DATA_BLOCK "DB23_AlarmProgram"   // DB23
{ S7_Optimized_Access := 'FALSE' }
AUTHOR : Robopac
VERSION : 0.0
// stored: AutoNumber false, IsOnlyStoredInLoadMemory false, IsWriteProtectedInAS false
   VAR RETAIN
      dbx0_0 : Bool := FALSE;   // Alarm 1: Pressure switch (Technoplat)
      dbx0_1 : Bool := FALSE;   // Alarm 2: Door open request (Technoplat)
      dbx0_2 : Bool := FALSE;   // Alarm 3: Emergency push button (Technoplat)
      dbx0_3 : Bool := FALSE;   // Alarm 4: Thermic alarm (Technoplat)
      dbx0_4 : Bool := FALSE;   // Alarm 5: Fault inverters (Technoplat)
      dbx0_5 : Bool := FALSE;   // Alarm 6: Motor start missing (Technoplat)
      dbx0_6 : Bool := FALSE;   // Alarm 7: Stop cycle by operator (Technoplat)
      dbx0_7 : Bool := FALSE;   // Alarm 8: Film ended or broken (Technoplat)
      dbx1_0 : Bool := FALSE;   // Alarm 9: Machine table not in phase (Technoplat)
      dbx1_1 : Bool := FALSE;   // Alarm 10: The spool carriage encoder is not running (Technoplat)
      dbx1_2 : Bool := FALSE;   // Alarm 11: Table encoder not working well
      dbx1_3 : Bool := FALSE;   // Alarm 12: Overspeed for table rotation (Technoplat)
      dbx1_4 : Bool := FALSE;   // Alarm 13: Phase table sensor lost (Technoplat)
      dbx1_5 : Bool := FALSE;   // Alarm 14: table deceleration not correct (Technoplat)
      dbx1_6 : Bool := FALSE;   // Alarm 15: Pressure plate not up (Pressure plate)
      dbx1_7 : Bool := FALSE;   // Alarm 16: Timeout for pressure plate upward/downward (Pressure plate)
      dbx2_0 : Bool := FALSE;   // Alarm 17: Pallet lifter not down (Lifter)
      dbx2_1 : Bool := FALSE;   // Alarm 18: Timeout for pallet lifter upward/downward (Lifter)
      dbx2_2 : Bool := FALSE;   // Alarm 19: Wrong data program for the pallet on the machine (Technoplat)
      dbx2_3 : Bool := FALSE;   // Alarm 20: Sysdata error (Technoplat)
      dbx2_4 : Bool := FALSE;   // Alarm 21: Spool carriage not down (Technoplat)
      dbx2_5 : Bool := FALSE;   // Alarm 22: Pressure plate positioning lost during rotation
      dbx2_6 : Bool := FALSE;   // Alarm 23:
      dbx2_7 : Bool := FALSE;   // Alarm 24: Emergency on infeed safety barrier (Barrier)
      dbx3_0 : Bool := FALSE;   // Alarm 25: Emergency on outfeed safety barrier (Barrier)
      dbx3_1 : Bool := FALSE;   // Alarm 26: Safety barrier excluded in automatic mode (Barrier)
      dbx3_2 : Bool := FALSE;   // Alarm 27: Timeout for rope unit open/close (Rope unit)
      dbx3_3 : Bool := FALSE;   // Alarm 28: Timeout for full rope unit open/close (Rope unit)
      dbx3_4 : Bool := FALSE;   // Alarm 29:
      dbx3_5 : Bool := FALSE;   // Alarm 30: Profinet communication error
      dbx3_6 : Bool := FALSE;   // Alarm 31: Modbus communication error
      dbx3_7 : Bool := FALSE;   // Alarm 32:
      dbx4_0 : Bool := FALSE;   // Alarm 33: Pallet positioning released during table rotation (Conveyor
      dbx4_1 : Bool := FALSE;   // Alarm 34: Pallet in transit in infeed (Conveyor)
      dbx4_2 : Bool := FALSE;   // Alarm 35: Pallet in transit in outfeed (Conveyor)
      dbx4_3 : Bool := FALSE;   // Alarm 36: Wrong pallet positioning (Conveyor)
      dbx4_4 : Bool := FALSE;   // Alarm 37: Infeed ring rotation control engaged (Conveyor)
      dbx4_5 : Bool := FALSE;   // Alarm 38: Outfeed ring rotation control engaged (Conveyor)
      dbx4_6 : Bool := FALSE;   // Alarm 39: Technoplat table not in load phase
      dbx4_7 : Bool := FALSE;   // Alarm 40: Technoplat table not in unload phase
      dbx5_0 : Bool := FALSE;   // Alarm 41: Contrast carriage not back
      dbx5_1 : Bool := FALSE;   // Alarm 42: Timeout contrast carriage forward/backward
      dbx5_2 : Bool := FALSE;   // Alarm 43: Clamp not closed (Clamp)
      dbx5_3 : Bool := FALSE;   // Alarm 44: Welder contrast not down (Clamp)
      dbx5_4 : Bool := FALSE;   // Alarm 45: Welder unit not down (Clamp)
      dbx5_5 : Bool := FALSE;   // Alarm 46: Clamp not down (Clamp)
      dbx5_6 : Bool := FALSE;   // Alarm 47: Welder contrast not up (Clamp)
      dbx5_7 : Bool := FALSE;   // Alarm 48: Timeout for clamp open/close (Clamp)
      dbx6_0 : Bool := FALSE;   // Alarm 49: Timeout for clamp upward/downward (Clamp)
      dbx6_1 : Bool := FALSE;   // Alarm 50: Timeout for welder contrast upward/downward (Clamp)
      dbx6_2 : Bool := FALSE;   // Alarm 51: Timeout for welder unit upward/downward (Clamp)
      dbx6_3 : Bool := FALSE;   // Alarm 52: Check the welder circuit (Clamp)
      dbx6_4 : Bool := FALSE;   // Alarm 53: Welder and cut unit not backward (Clamp)
      dbx6_5 : Bool := FALSE;   // Alarm 54: Timeout for welder and cut unit forward/backward (Clamp)
      dbx6_6 : Bool := FALSE;   // Alarm 55: Timeout for clamp carriage forward/backward (Clamp)
      dbx6_7 : Bool := FALSE;   // Alarm 56: Clamp carriage not backward (Clamp)
      dbx7_0 : Bool := FALSE;   // Alarm 57: Top carriage not up (Top)
      dbx7_1 : Bool := FALSE;   // Alarm 58: Top carriage not backward (Top)
      dbx7_2 : Bool := FALSE;   // Alarm 59: Top cutter not backward (Top)
      dbx7_3 : Bool := FALSE;   // Alarm 60: Clamp to pull top film not open (Top)
      dbx7_4 : Bool := FALSE;   // Alarm 61: Clamp to block top film not closed (Top)
      dbx7_5 : Bool := FALSE;   // Alarm 62: Top carriage not in position (Top)
      dbx7_6 : Bool := FALSE;   // Alarm 63: Top carriage not inside top film cut area (Top)
      dbx7_7 : Bool := FALSE;   // Alarm 64: Safety for top carriage position (Top)
      dbx8_0 : Bool := FALSE;   // Alarm 65: Timeout for top cutter (Top)
      dbx8_1 : Bool := FALSE;   // Alarm 66: Timeout for clamp to pull top film (Top)
      dbx8_2 : Bool := FALSE;   // Alarm 67: Timeout for clamp to block top film (Top)
      dbx8_3 : Bool := FALSE;   // Alarm 68: Top film ended or broken (Top)
      dbx8_4 : Bool := FALSE;   // Alarm 69: Infeed safety for top carriage up/down (Top)
      dbx8_5 : Bool := FALSE;   // Alarm 70: Outfeed safety for top carriage up/down (Top)
      dbx8_6 : Bool := FALSE;   // Alarm 71: Clamp to blok top film not open (Top)
      dbx8_7 : Bool := FALSE;   // Alarm 72: Top rele' brake broken (Top)
      dbx9_0 : Bool := FALSE;   // Alarm 73: Top not in position (Top inside signal)
      dbx9_1 : Bool := FALSE;   // Alarm 74: LIFTER POS.2 EXTRASTROKE UP
      dbx9_2 : Bool := FALSE;   // Alarm 75: LIFTER POS.2 FOOT SAFETY
      dbx9_3 : Bool := FALSE;   // Alarm 76: LIFTER POS.2 TIMEOUT CONVEYOR
      dbx9_4 : Bool := FALSE;   // Alarm 77: LIFTER POS.2 TIMEOUT UPSTROKE
      dbx9_5 : Bool := FALSE;   // Alarm 78: LIFTER POS.2 TIMEOUT DOWNSTROKE
      dbx9_6 : Bool := FALSE;   // Alarm 79: LABEL FAULT
      dbx9_7 : Bool := FALSE;   // Alarm 80: Label not in home position with table rotation
      dbx10_0 : Bool := FALSE;   // Alarm 81: Fire door not open during pallet transit
      dbx10_1 : Bool := FALSE;   // Alarm 82:
      dbx10_2 : Bool := FALSE;   // Alarm 83:
      dbx10_3 : Bool := FALSE;   // Alarm 84:
      dbx10_4 : Bool := FALSE;   // Alarm 85:
      dbx10_5 : Bool := FALSE;   // Alarm 86:
      dbx10_6 : Bool := FALSE;   // Alarm 87:
      dbx10_7 : Bool := FALSE;   // Alarm 88:
      dbx11_0 : Bool := FALSE;   // Alarm 89:
      dbx11_1 : Bool := FALSE;   // Alarm 90:
      dbx11_2 : Bool := FALSE;   // Alarm 91:
      dbx11_3 : Bool := FALSE;   // Alarm 92:
      dbx11_4 : Bool := FALSE;   // Alarm 93:
      dbx11_5 : Bool := FALSE;   // Alarm 94:
      dbx11_6 : Bool := FALSE;   // Alarm 95:
      dbx11_7 : Bool := FALSE;   // Alarm 96:
      dbx12_0 : Bool := FALSE;   // Alarm 97:
      dbx12_1 : Bool := FALSE;   // Alarm 98:
      dbx12_2 : Bool := FALSE;   // Alarm 99:
      dbx12_3 : Bool := FALSE;   // Alarm 100:
      dbx12_4 : Bool := FALSE;   // Alarm 101:
      dbx12_5 : Bool := FALSE;   // Alarm 102:
      dbx12_6 : Bool := FALSE;   // Alarm 103:
      dbx12_7 : Bool := FALSE;   // Alarm 104:
      dbx13_0 : Bool := FALSE;   // Alarm 105:
      dbx13_1 : Bool := FALSE;   // Alarm 106:
      dbx13_2 : Bool := FALSE;   // Alarm 107:
      dbx13_3 : Bool := FALSE;   // Alarm 108:
      dbx13_4 : Bool := FALSE;   // Alarm 109:
      dbx13_5 : Bool := FALSE;   // Alarm 110:
      dbx13_6 : Bool := FALSE;   // Alarm 111:
      dbx13_7 : Bool := FALSE;   // Alarm 112:
      dbx14_0 : Bool := FALSE;   // Alarm 113:
      dbx14_1 : Bool := FALSE;   // Alarm 114:
      dbx14_2 : Bool := FALSE;   // Alarm 115:
      dbx14_3 : Bool := FALSE;   // Alarm 116:
      dbx14_4 : Bool := FALSE;   // Alarm 117:
      dbx14_5 : Bool := FALSE;   // Alarm 118:
      dbx14_6 : Bool := FALSE;   // Alarm 119:
      dbx14_7 : Bool := FALSE;   // Alarm 120:
      dbx15_0 : Bool := FALSE;   // Alarm 121:
      dbx15_1 : Bool := FALSE;   // Alarm 122:
      dbx15_2 : Bool := FALSE;   // Alarm 123:
      dbx15_3 : Bool := FALSE;   // Alarm 124:
      dbx15_4 : Bool := FALSE;   // Alarm 125:
      dbx15_5 : Bool := FALSE;   // Alarm 126:
      dbx15_6 : Bool := FALSE;   // Alarm 127:
      dbx15_7 : Bool := FALSE;   // Alarm 128:
      dbx16_0 : Bool := FALSE;   // Alarm 129:
      dbx16_1 : Bool := FALSE;   // Alarm 130:
      dbx16_2 : Bool := FALSE;   // Alarm 131:
      dbx16_3 : Bool := FALSE;   // Alarm 132:
      dbx16_4 : Bool := FALSE;   // Alarm 133:
      dbx16_5 : Bool := FALSE;   // Alarm 134:
      dbx16_6 : Bool := FALSE;   // Alarm 135:
      dbx16_7 : Bool := FALSE;   // Alarm 136:
      dbx17_0 : Bool := FALSE;   // Alarm 137:
      dbx17_1 : Bool := FALSE;   // Alarm 138:
      dbx17_2 : Bool := FALSE;   // Alarm 139:
      dbx17_3 : Bool := FALSE;   // Alarm 140:
      dbx17_4 : Bool := FALSE;   // Alarm 141:
      dbx17_5 : Bool := FALSE;   // Alarm 142:
      dbx17_6 : Bool := FALSE;   // Alarm 143:
      dbx17_7 : Bool := FALSE;   // Alarm 144:
      dbx18_0 : Bool := FALSE;   // Alarm 145:
      dbx18_1 : Bool := FALSE;   // Alarm 146:
      dbx18_2 : Bool := FALSE;   // Alarm 147:
      dbx18_3 : Bool := FALSE;   // Alarm 148:
      dbx18_4 : Bool := FALSE;   // Alarm 149:
      dbx18_5 : Bool := FALSE;   // Alarm 150:
      dbx18_6 : Bool := FALSE;   // Alarm 151:
      dbx18_7 : Bool := FALSE;   // Alarm 152:
      dbx19_0 : Bool := FALSE;   // Alarm 153:
      dbx19_1 : Bool := FALSE;   // Alarm 154:
      dbx19_2 : Bool := FALSE;   // Alarm 155:
      dbx19_3 : Bool := FALSE;   // Alarm 156:
      dbx19_4 : Bool := FALSE;   // Alarm 157:
      dbx19_5 : Bool := FALSE;   // Alarm 158:
      dbx19_6 : Bool := FALSE;   // Alarm 159:
      dbx19_7 : Bool := FALSE;   // Alarm 160:
      dbx20_0 : Bool := FALSE;   // Alarm 161:
      dbx20_1 : Bool := FALSE;   // Alarm 162:
      dbx20_2 : Bool := FALSE;   // Alarm 163:
      dbx20_3 : Bool := FALSE;   // Alarm 164:
      dbx20_4 : Bool := FALSE;   // Alarm 165:
      dbx20_5 : Bool := FALSE;   // Alarm 166:
      dbx20_6 : Bool := FALSE;   // Alarm 167:
      dbx20_7 : Bool := FALSE;   // Alarm 168:
      dbx21_0 : Bool := FALSE;   // Alarm 169:
      dbx21_1 : Bool := FALSE;   // Alarm 170:
      dbx21_2 : Bool := FALSE;   // Alarm 171:
      dbx21_3 : Bool := FALSE;   // Alarm 172:
      dbx21_4 : Bool := FALSE;   // Alarm 173:
      dbx21_5 : Bool := FALSE;   // Alarm 174:
      dbx21_6 : Bool := FALSE;   // Alarm 175:
      dbx21_7 : Bool := FALSE;   // Alarm 176:
      dbx22_0 : Bool := FALSE;   // Alarm 177:
      dbx22_1 : Bool := FALSE;   // Alarm 178:
      dbx22_2 : Bool := FALSE;   // Alarm 179:
      dbx22_3 : Bool := FALSE;   // Alarm 180:
      dbx22_4 : Bool := FALSE;   // Alarm 181:
      dbx22_5 : Bool := FALSE;   // Alarm 182:
      dbx22_6 : Bool := FALSE;   // Alarm 183:
      dbx22_7 : Bool := FALSE;   // Alarm 184:
      dbx23_0 : Bool := FALSE;   // Alarm 185:
      dbx23_1 : Bool := FALSE;   // Alarm 186:
      dbx23_2 : Bool := FALSE;   // Alarm 187:
      dbx23_3 : Bool := FALSE;   // Alarm 188:
      dbx23_4 : Bool := FALSE;   // Alarm 189:
      dbx23_5 : Bool := FALSE;   // Alarm 190:
      dbx23_6 : Bool := FALSE;   // Alarm 191:
      dbx23_7 : Bool := FALSE;   // Alarm 192:
      dbx24_0 : Bool := FALSE;   // Alarm 193:
      dbx24_1 : Bool := FALSE;   // Alarm 194:
      dbx24_2 : Bool := FALSE;   // Alarm 195:
      dbx24_3 : Bool := FALSE;   // Alarm 196:
      dbx24_4 : Bool := FALSE;   // Alarm 197:
      dbx24_5 : Bool := FALSE;   // Alarm 198:
      dbx24_6 : Bool := FALSE;   // Alarm 199:
      dbx24_7 : Bool := FALSE;   // Alarm 200:
      dbx25_0 : Bool := FALSE;   // Alarm 201:
      dbx25_1 : Bool := FALSE;   // Alarm 202:
      dbx25_2 : Bool := FALSE;   // Alarm 203:
      dbx25_3 : Bool := FALSE;   // Alarm 204:
      dbx25_4 : Bool := FALSE;   // Alarm 205:
      dbx25_5 : Bool := FALSE;   // Alarm 206:
      dbx25_6 : Bool := FALSE;   // Alarm 207:
      dbx25_7 : Bool := FALSE;   // Alarm 208:
      dbx26_0 : Bool := FALSE;   // Warning 1: %10 Prestretch film on spool carriage (Technoplat)
      dbx26_1 : Bool := FALSE;   // Warning 2:
      dbx26_2 : Bool := FALSE;   // Warning 3: Request to reset encoder on spool carriage (Technoplat)
      dbx26_3 : Bool := FALSE;   // Warning 4:
      dbx26_4 : Bool := FALSE;   // Warning 5: Request to reset encoder on table rotation (Technoplat)
      dbx26_5 : Bool := FALSE;   // Warning 6:
      dbx26_6 : Bool := FALSE;   // Warning 7:
      dbx26_7 : Bool := FALSE;   // Warning 8: Fire door closing request
      dbx27_0 : Bool := FALSE;   // Warning 9: Timeout for door opening
      dbx27_1 : Bool := FALSE;   // Warning 10:
      dbx27_2 : Bool := FALSE;   // Warning 11:
      dbx27_3 : Bool := FALSE;   // Warning 12:
      dbx27_4 : Bool := FALSE;   // Warning 13:
      dbx27_5 : Bool := FALSE;   // Warning 14:
      dbx27_6 : Bool := FALSE;   // Warning 15:
      dbx27_7 : Bool := FALSE;   // Warning 16:
      dbx28_0 : Bool := FALSE;   // Warning 17:
      dbx28_1 : Bool := FALSE;   // Warning 18:
      dbx28_2 : Bool := FALSE;   // Warning 19:
      dbx28_3 : Bool := FALSE;   // Warning 20:
      dbx28_4 : Bool := FALSE;   // Warning 21:
      dbx28_5 : Bool := FALSE;   // Warning 22:
      dbx28_6 : Bool := FALSE;   // Warning 23:
      dbx28_7 : Bool := FALSE;   // Warning 24:
      dbx29_0 : Bool := FALSE;   // Warning 25:
      dbx29_1 : Bool := FALSE;   // Warning 26:
      dbx29_2 : Bool := FALSE;   // Warning 27:
      dbx29_3 : Bool := FALSE;   // Warning 28:
      dbx29_4 : Bool := FALSE;   // Warning 29:
      dbx29_5 : Bool := FALSE;   // Warning 30:
      dbx29_6 : Bool := FALSE;   // Warning 31:
      dbx29_7 : Bool := FALSE;   // Warning 32:
   END_VAR
BEGIN
END_DATA_BLOCK

DATA_BLOCK "DB240_Program10"   // DB240
{ S7_Optimized_Access := 'FALSE' }
AUTHOR : Robopac
VERSION : 0.0
// stored: AutoNumber false, IsOnlyStoredInLoadMemory false, IsWriteProtectedInAS false
   VAR RETAIN
      Program10 { S7_SetPoint := 'True'} : "DatiProgramma";
   END_VAR
BEGIN
   Program10.Wrapping := TRUE;
   Program10.TopLenght := 500;
   Program10.TopRelease := 0;
   Program10.TopDown := 0;
   Program10.Top := 4;
   Program10.PressurePTime := 0;
   Program10.LifterTime := 0;
   Program10.RevOverContrast := 1;
   Program10.RopeEndCycle := 16#02;
   Program10.Spare4 := 16#01;
   Program10.RopeTime := 1500;
   Program10.RevOverClamp := 1;
   Program10.FilmForceFinalRev := 10;
   Program10.FilmPrestretchFinalRev := 100;
   Program10.ArmSpeed := 100;
   Program10.CarriageDown4Top := 500;
   Program10.TopDownTime := 1500;
   Program10.LapsUnderTop := 0;
   Program10.Spare6 := 0;
   Program10.Spare7 := 0;
   Program10.Spare8 := 0;
   Program10.Spare9 := 0;
   Program10.Spare10 := 0;
   Program10.Spare11 := 0;
   Program10.Spare12 := 0;
   Program10.Overlap0_1 := 0;
   Program10.Height1 := 130;
   Program10.Landmark1 := FALSE;
   Program10.Lifter1 := FALSE;
   Program10.SpareBit1H1 := FALSE;
   Program10.Airblower1 := TRUE;
   Program10.NextStep1 := TRUE;
   Program10.PressureP1 := TRUE;
   Program10.SpareByte2H1 := 16#00;
   Program10.Revolution1 := 1;
   Program10.RopeUnit1_1 := 16#01;
   Program10.RopeUnit1_2 := 16#01;
   Program10.FilmForce1 := 5;
   Program10.FilmPrestretch1 := 200;
   Program10.Spare3H1 := 0;
   Program10.Spare49 := 0;
   Program10.Spare50 := 0;
   Program10.Spare51 := 0;
   Program10.Spare52 := 0;
   Program10.Spare53 := 0;
   Program10.Overlap1_2 := 0;
   Program10.Height2 := 50;
   Program10.Landmark2 := FALSE;
   Program10.Lifter2 := FALSE;
   Program10.SpareBit1H2 := FALSE;
   Program10.Airblower2 := TRUE;
   Program10.NextStep2 := TRUE;
   Program10.PressureP2 := TRUE;
   Program10.SpareByte2H2 := 16#00;
   Program10.Revolution2 := 1;
   Program10.RopeUnit2_1 := 16#01;
   Program10.RopeUnit2_2 := 16#01;
   Program10.FilmForce2 := 20;
   Program10.FilmPrestretch2 := 200;
   Program10.Spare3H2 := 0;
   Program10.Spare54 := 0;
   Program10.Spare55 := 0;
   Program10.Spare56 := 0;
   Program10.Spare57 := 0;
   Program10.Spare58 := 0;
   Program10.Overlap2_3 := 100;
   Program10.Height3 := -50;
   Program10.Landmark3 := TRUE;
   Program10.Lifter3 := FALSE;
   Program10.SpareBit1H3 := FALSE;
   Program10.Airblower3 := TRUE;
   Program10.NextStep3 := TRUE;
   Program10.PressureP3 := TRUE;
   Program10.SpareByte2H3 := 16#00;
   Program10.Revolution3 := 2;
   Program10.RopeUnit3_1 := 16#01;
   Program10.RopeUnit3_2 := 16#01;
   Program10.FilmForce3 := 30;
   Program10.FilmPrestretch3 := 200;
   Program10.Spare3H3 := 0;
   Program10.Spare59 := 0;
   Program10.Spare60 := 0;
   Program10.Spare61 := 380;
   Program10.Spare62 := 2800;
   Program10.Spare63 := 0;
   Program10.Overlap3_4 := 100;
   Program10.Height4 := 100;
   Program10.Landmark4 := FALSE;
   Program10.Lifter4 := FALSE;
   Program10.SpareBit1H4 := FALSE;
   Program10.Airblower4 := TRUE;
   Program10.NextStep4 := TRUE;
   Program10.PressureP4 := TRUE;
   Program10.SpareByte2H4 := 16#00;
   Program10.Revolution4 := 3;
   Program10.RopeUnit4_1 := 16#02;
   Program10.RopeUnit4_2 := 16#02;
   Program10.FilmForce4 := 30;
   Program10.FilmPrestretch4 := 200;
   Program10.Spare3H4 := 0;
   Program10.Spare64 := 0;
   Program10.Spare65 := 0;
   Program10.Spare66 := 0;
   Program10.Spare67 := 0;
   Program10.Spare68 := 0;
   Program10.Overlap4_5 := 0;
   Program10.Height5 := 50;
   Program10.Landmark5 := FALSE;
   Program10.Lifter5 := FALSE;
   Program10.SpareBit1H5 := FALSE;
   Program10.Airblower5 := TRUE;
   Program10.NextStep5 := FALSE;
   Program10.PressureP5 := FALSE;
   Program10.SpareByte2H5 := 16#00;
   Program10.Revolution5 := 1;
   Program10.RopeUnit5_1 := 16#01;
   Program10.RopeUnit5_2 := 16#01;
   Program10.FilmForce5 := 30;
   Program10.FilmPrestretch5 := 200;
   Program10.Spare3H5 := 0;
   Program10.Spare69 := 0;
   Program10.Spare70 := 0;
   Program10.Spare71 := 0;
   Program10.Spare72 := 0;
   Program10.Spare73 := 0;
   Program10.Overlap5_6 := 100;
   Program10.Height6 := 50;
   Program10.Landmark6 := FALSE;
   Program10.Lifter6 := FALSE;
   Program10.SpareBit1H6 := FALSE;
   Program10.Airblower6 := TRUE;
   Program10.NextStep6 := FALSE;
   Program10.PressureP6 := FALSE;
   Program10.SpareByte2H6 := 16#00;
   Program10.Revolution6 := 2;
   Program10.RopeUnit6_1 := 16#02;
   Program10.RopeUnit6_2 := 16#01;
   Program10.FilmForce6 := 20;
   Program10.FilmPrestretch6 := 200;
   Program10.Spare3H6 := 0;
   Program10.Spare74 := 0;
   Program10.Spare75 := 0;
   Program10.Spare76 := 0;
   Program10.Spare77 := 0;
   Program10.Spare78 := 0;
   Program10.Overlap6_7 := 0;
   Program10.Height7 := 0;
   Program10.Landmark7 := FALSE;
   Program10.Lifter7 := FALSE;
   Program10.SpareBit1H7 := FALSE;
   Program10.Airblower7 := FALSE;
   Program10.NextStep7 := TRUE;
   Program10.PressureP7 := FALSE;
   Program10.SpareByte2H7 := 16#00;
   Program10.Revolution7 := 1;
   Program10.RopeUnit7_1 := 16#01;
   Program10.RopeUnit7_2 := 16#01;
   Program10.FilmForce7 := 0;
   Program10.FilmPrestretch7 := 100;
   Program10.Spare3H7 := 0;
   Program10.Spare79 := 0;
   Program10.Spare80 := 0;
   Program10.Spare81 := 0;
   Program10.Spare82 := 0;
   Program10.Spare83 := 0;
   Program10.Overlap7_8 := 0;
   Program10.Height8 := 0;
   Program10.Landmark8 := FALSE;
   Program10.Lifter8 := FALSE;
   Program10.SpareBit1H8 := FALSE;
   Program10.Airblower8 := FALSE;
   Program10.NextStep8 := TRUE;
   Program10.PressureP8 := FALSE;
   Program10.SpareByte2H8 := 16#00;
   Program10.Revolution8 := 1;
   Program10.RopeUnit8_1 := 16#01;
   Program10.RopeUnit8_2 := 16#01;
   Program10.FilmForce8 := 0;
   Program10.FilmPrestretch8 := 100;
   Program10.Spare3H8 := 0;
   Program10.Spare84 := 0;
   Program10.Spare85 := 0;
   Program10.Spare86 := 0;
   Program10.Spare87 := 0;
   Program10.Spare88 := 0;
   Program10.Overlap8_9 := 0;
   Program10.Height9 := 0;
   Program10.Landmark9 := FALSE;
   Program10.Lifter9 := FALSE;
   Program10.SpareBit1H9 := FALSE;
   Program10.Airblower9 := FALSE;
   Program10.NextStep9 := TRUE;
   Program10.PressureP9 := FALSE;
   Program10.SpareByte2H9 := 16#00;
   Program10.Revolution9 := 1;
   Program10.RopeUnit9_1 := 16#01;
   Program10.RopeUnit9_2 := 16#01;
   Program10.FilmForce9 := 0;
   Program10.FilmPrestretch9 := 100;
   Program10.Spare3H9 := 0;
   Program10.Spare89 := 0;
   Program10.Spare90 := 0;
   Program10.Spare91 := 0;
   Program10.Spare92 := 0;
   Program10.Spare93 := 0;
   Program10.Overlap9_10 := 0;
   Program10.Height10 := 0;
   Program10.Landmark10 := FALSE;
   Program10.Lifter10 := FALSE;
   Program10.SpareBit1H10 := FALSE;
   Program10.Airblower10 := FALSE;
   Program10.NextStep10 := FALSE;
   Program10.PressureP10 := FALSE;
   Program10.SpareByte2H10 := 16#00;
   Program10.Revolution10 := 1;
   Program10.RopeUnit10_1 := 16#01;
   Program10.RopeUnit10_2 := 16#01;
   Program10.FilmForce10 := 0;
   Program10.FilmPrestretch10 := 100;
   Program10.Spare3H10 := 0;
   Program10.Spare94 := 0;
   Program10.Spare95 := 0;
   Program10.Spare96 := 0;
   Program10.Spare97 := 0;
   Program10.Spare98 := 0;
   Program10.Overlap10_11 := 0;
   Program10.Height11 := 0;
   Program10.Landmark11 := FALSE;
   Program10.Lifter11 := FALSE;
   Program10.SpareBit1H11 := FALSE;
   Program10.Airblower11 := FALSE;
   Program10.NextStep11 := TRUE;
   Program10.PressureP11 := FALSE;
   Program10.SpareByte2H11 := 16#00;
   Program10.Revolution11 := 1;
   Program10.RopeUnit11_1 := 16#01;
   Program10.RopeUnit11_2 := 16#01;
   Program10.FilmForce11 := 0;
   Program10.FilmPrestretch11 := 100;
   Program10.Spare3H11 := 0;
   Program10.Spare99 := 0;
   Program10.Spare100 := 0;
   Program10.Spare101 := 0;
   Program10.Spare102 := 0;
   Program10.Spare103 := 0;
   Program10.Overlap11_12 := 0;
   Program10.Height12 := 0;
   Program10.Landmark12 := FALSE;
   Program10.Lifter12 := FALSE;
   Program10.SpareBit1H12 := FALSE;
   Program10.Airblower12 := FALSE;
   Program10.NextStep12 := FALSE;
   Program10.PressureP12 := FALSE;
   Program10.SpareByte2H12 := 16#00;
   Program10.Revolution12 := 1;
   Program10.RopeUnit12_1 := 16#01;
   Program10.RopeUnit12_2 := 16#01;
   Program10.FilmForce12 := 0;
   Program10.FilmPrestretch12 := 100;
   Program10.Spare3H12 := 0;
   Program10.Spare104 := 0;
   Program10.Spare105 := 0;
   Program10.Spare106 := 0;
   Program10.Spare107 := 0;
   Program10.Spare108 := 0;
END_DATA_BLOCK

DATA_BLOCK "DB241_Program9"   // DB241
{ S7_Optimized_Access := 'FALSE' }
AUTHOR : Robopac
VERSION : 0.0
// stored: AutoNumber false, IsOnlyStoredInLoadMemory false, IsWriteProtectedInAS false
   VAR RETAIN
      Program9 { S7_SetPoint := 'True'} : "DatiProgramma";
   END_VAR
BEGIN
   Program9.Wrapping := TRUE;
   Program9.TopLenght := 500;
   Program9.TopRelease := 0;
   Program9.TopDown := 0;
   Program9.Top := 4;
   Program9.PressurePTime := 0;
   Program9.LifterTime := 0;
   Program9.RevOverContrast := 1;
   Program9.RopeEndCycle := 16#02;
   Program9.Spare4 := 16#01;
   Program9.RopeTime := 1500;
   Program9.RevOverClamp := 1;
   Program9.FilmForceFinalRev := 10;
   Program9.FilmPrestretchFinalRev := 100;
   Program9.ArmSpeed := 100;
   Program9.CarriageDown4Top := 500;
   Program9.TopDownTime := 1500;
   Program9.LapsUnderTop := 0;
   Program9.Spare6 := 0;
   Program9.Spare7 := 0;
   Program9.Spare8 := 0;
   Program9.Spare9 := 0;
   Program9.Spare10 := 0;
   Program9.Spare11 := 0;
   Program9.Spare12 := 0;
   Program9.Overlap0_1 := 0;
   Program9.Height1 := 130;
   Program9.Landmark1 := FALSE;
   Program9.Lifter1 := FALSE;
   Program9.SpareBit1H1 := FALSE;
   Program9.Airblower1 := TRUE;
   Program9.NextStep1 := TRUE;
   Program9.PressureP1 := TRUE;
   Program9.SpareByte2H1 := 16#00;
   Program9.Revolution1 := 1;
   Program9.RopeUnit1_1 := 16#01;
   Program9.RopeUnit1_2 := 16#01;
   Program9.FilmForce1 := 5;
   Program9.FilmPrestretch1 := 200;
   Program9.Spare3H1 := 0;
   Program9.Spare49 := 0;
   Program9.Spare50 := 0;
   Program9.Spare51 := 0;
   Program9.Spare52 := 0;
   Program9.Spare53 := 0;
   Program9.Overlap1_2 := 0;
   Program9.Height2 := 50;
   Program9.Landmark2 := FALSE;
   Program9.Lifter2 := FALSE;
   Program9.SpareBit1H2 := FALSE;
   Program9.Airblower2 := TRUE;
   Program9.NextStep2 := TRUE;
   Program9.PressureP2 := TRUE;
   Program9.SpareByte2H2 := 16#00;
   Program9.Revolution2 := 1;
   Program9.RopeUnit2_1 := 16#01;
   Program9.RopeUnit2_2 := 16#01;
   Program9.FilmForce2 := 20;
   Program9.FilmPrestretch2 := 200;
   Program9.Spare3H2 := 0;
   Program9.Spare54 := 0;
   Program9.Spare55 := 0;
   Program9.Spare56 := 0;
   Program9.Spare57 := 0;
   Program9.Spare58 := 0;
   Program9.Overlap2_3 := 100;
   Program9.Height3 := -50;
   Program9.Landmark3 := TRUE;
   Program9.Lifter3 := FALSE;
   Program9.SpareBit1H3 := FALSE;
   Program9.Airblower3 := TRUE;
   Program9.NextStep3 := TRUE;
   Program9.PressureP3 := TRUE;
   Program9.SpareByte2H3 := 16#00;
   Program9.Revolution3 := 2;
   Program9.RopeUnit3_1 := 16#01;
   Program9.RopeUnit3_2 := 16#01;
   Program9.FilmForce3 := 30;
   Program9.FilmPrestretch3 := 200;
   Program9.Spare3H3 := 0;
   Program9.Spare59 := 0;
   Program9.Spare60 := 0;
   Program9.Spare61 := 380;
   Program9.Spare62 := 2800;
   Program9.Spare63 := 0;
   Program9.Overlap3_4 := 100;
   Program9.Height4 := 100;
   Program9.Landmark4 := FALSE;
   Program9.Lifter4 := FALSE;
   Program9.SpareBit1H4 := FALSE;
   Program9.Airblower4 := TRUE;
   Program9.NextStep4 := TRUE;
   Program9.PressureP4 := TRUE;
   Program9.SpareByte2H4 := 16#00;
   Program9.Revolution4 := 3;
   Program9.RopeUnit4_1 := 16#02;
   Program9.RopeUnit4_2 := 16#02;
   Program9.FilmForce4 := 30;
   Program9.FilmPrestretch4 := 200;
   Program9.Spare3H4 := 0;
   Program9.Spare64 := 0;
   Program9.Spare65 := 0;
   Program9.Spare66 := 0;
   Program9.Spare67 := 0;
   Program9.Spare68 := 0;
   Program9.Overlap4_5 := 0;
   Program9.Height5 := 50;
   Program9.Landmark5 := FALSE;
   Program9.Lifter5 := FALSE;
   Program9.SpareBit1H5 := FALSE;
   Program9.Airblower5 := TRUE;
   Program9.NextStep5 := FALSE;
   Program9.PressureP5 := FALSE;
   Program9.SpareByte2H5 := 16#00;
   Program9.Revolution5 := 1;
   Program9.RopeUnit5_1 := 16#01;
   Program9.RopeUnit5_2 := 16#01;
   Program9.FilmForce5 := 30;
   Program9.FilmPrestretch5 := 200;
   Program9.Spare3H5 := 0;
   Program9.Spare69 := 0;
   Program9.Spare70 := 0;
   Program9.Spare71 := 0;
   Program9.Spare72 := 0;
   Program9.Spare73 := 0;
   Program9.Overlap5_6 := 100;
   Program9.Height6 := 50;
   Program9.Landmark6 := FALSE;
   Program9.Lifter6 := FALSE;
   Program9.SpareBit1H6 := FALSE;
   Program9.Airblower6 := TRUE;
   Program9.NextStep6 := FALSE;
   Program9.PressureP6 := FALSE;
   Program9.SpareByte2H6 := 16#00;
   Program9.Revolution6 := 2;
   Program9.RopeUnit6_1 := 16#02;
   Program9.RopeUnit6_2 := 16#01;
   Program9.FilmForce6 := 20;
   Program9.FilmPrestretch6 := 200;
   Program9.Spare3H6 := 0;
   Program9.Spare74 := 0;
   Program9.Spare75 := 0;
   Program9.Spare76 := 0;
   Program9.Spare77 := 0;
   Program9.Spare78 := 0;
   Program9.Overlap6_7 := 0;
   Program9.Height7 := 0;
   Program9.Landmark7 := FALSE;
   Program9.Lifter7 := FALSE;
   Program9.SpareBit1H7 := FALSE;
   Program9.Airblower7 := FALSE;
   Program9.NextStep7 := TRUE;
   Program9.PressureP7 := FALSE;
   Program9.SpareByte2H7 := 16#00;
   Program9.Revolution7 := 1;
   Program9.RopeUnit7_1 := 16#01;
   Program9.RopeUnit7_2 := 16#01;
   Program9.FilmForce7 := 0;
   Program9.FilmPrestretch7 := 100;
   Program9.Spare3H7 := 0;
   Program9.Spare79 := 0;
   Program9.Spare80 := 0;
   Program9.Spare81 := 0;
   Program9.Spare82 := 0;
   Program9.Spare83 := 0;
   Program9.Overlap7_8 := 0;
   Program9.Height8 := 0;
   Program9.Landmark8 := FALSE;
   Program9.Lifter8 := FALSE;
   Program9.SpareBit1H8 := FALSE;
   Program9.Airblower8 := FALSE;
   Program9.NextStep8 := TRUE;
   Program9.PressureP8 := FALSE;
   Program9.SpareByte2H8 := 16#00;
   Program9.Revolution8 := 1;
   Program9.RopeUnit8_1 := 16#01;
   Program9.RopeUnit8_2 := 16#01;
   Program9.FilmForce8 := 0;
   Program9.FilmPrestretch8 := 100;
   Program9.Spare3H8 := 0;
   Program9.Spare84 := 0;
   Program9.Spare85 := 0;
   Program9.Spare86 := 0;
   Program9.Spare87 := 0;
   Program9.Spare88 := 0;
   Program9.Overlap8_9 := 0;
   Program9.Height9 := 0;
   Program9.Landmark9 := FALSE;
   Program9.Lifter9 := FALSE;
   Program9.SpareBit1H9 := FALSE;
   Program9.Airblower9 := FALSE;
   Program9.NextStep9 := TRUE;
   Program9.PressureP9 := FALSE;
   Program9.SpareByte2H9 := 16#00;
   Program9.Revolution9 := 1;
   Program9.RopeUnit9_1 := 16#01;
   Program9.RopeUnit9_2 := 16#01;
   Program9.FilmForce9 := 0;
   Program9.FilmPrestretch9 := 100;
   Program9.Spare3H9 := 0;
   Program9.Spare89 := 0;
   Program9.Spare90 := 0;
   Program9.Spare91 := 0;
   Program9.Spare92 := 0;
   Program9.Spare93 := 0;
   Program9.Overlap9_10 := 0;
   Program9.Height10 := 0;
   Program9.Landmark10 := FALSE;
   Program9.Lifter10 := FALSE;
   Program9.SpareBit1H10 := FALSE;
   Program9.Airblower10 := FALSE;
   Program9.NextStep10 := FALSE;
   Program9.PressureP10 := FALSE;
   Program9.SpareByte2H10 := 16#00;
   Program9.Revolution10 := 1;
   Program9.RopeUnit10_1 := 16#01;
   Program9.RopeUnit10_2 := 16#01;
   Program9.FilmForce10 := 0;
   Program9.FilmPrestretch10 := 100;
   Program9.Spare3H10 := 0;
   Program9.Spare94 := 0;
   Program9.Spare95 := 0;
   Program9.Spare96 := 0;
   Program9.Spare97 := 0;
   Program9.Spare98 := 0;
   Program9.Overlap10_11 := 0;
   Program9.Height11 := 0;
   Program9.Landmark11 := FALSE;
   Program9.Lifter11 := FALSE;
   Program9.SpareBit1H11 := FALSE;
   Program9.Airblower11 := FALSE;
   Program9.NextStep11 := TRUE;
   Program9.PressureP11 := FALSE;
   Program9.SpareByte2H11 := 16#00;
   Program9.Revolution11 := 1;
   Program9.RopeUnit11_1 := 16#01;
   Program9.RopeUnit11_2 := 16#01;
   Program9.FilmForce11 := 0;
   Program9.FilmPrestretch11 := 100;
   Program9.Spare3H11 := 0;
   Program9.Spare99 := 0;
   Program9.Spare100 := 0;
   Program9.Spare101 := 0;
   Program9.Spare102 := 0;
   Program9.Spare103 := 0;
   Program9.Overlap11_12 := 0;
   Program9.Height12 := 0;
   Program9.Landmark12 := FALSE;
   Program9.Lifter12 := FALSE;
   Program9.SpareBit1H12 := FALSE;
   Program9.Airblower12 := FALSE;
   Program9.NextStep12 := FALSE;
   Program9.PressureP12 := FALSE;
   Program9.SpareByte2H12 := 16#00;
   Program9.Revolution12 := 1;
   Program9.RopeUnit12_1 := 16#01;
   Program9.RopeUnit12_2 := 16#01;
   Program9.FilmForce12 := 0;
   Program9.FilmPrestretch12 := 100;
   Program9.Spare3H12 := 0;
   Program9.Spare104 := 0;
   Program9.Spare105 := 0;
   Program9.Spare106 := 0;
   Program9.Spare107 := 0;
   Program9.Spare108 := 0;
END_DATA_BLOCK

DATA_BLOCK "DB242_Program8"   // DB242
{ S7_Optimized_Access := 'FALSE' }
AUTHOR : Robopac
VERSION : 0.0
// stored: AutoNumber false, IsOnlyStoredInLoadMemory false, IsWriteProtectedInAS false
   VAR RETAIN
      Program8 { S7_SetPoint := 'True'} : "DatiProgramma";
   END_VAR
BEGIN
   Program8.Wrapping := TRUE;
   Program8.TopLenght := 500;
   Program8.TopRelease := 0;
   Program8.TopDown := 0;
   Program8.Top := 4;
   Program8.PressurePTime := 0;
   Program8.LifterTime := 0;
   Program8.RevOverContrast := 1;
   Program8.RopeEndCycle := 16#02;
   Program8.Spare4 := 16#01;
   Program8.RopeTime := 1500;
   Program8.RevOverClamp := 1;
   Program8.FilmForceFinalRev := 10;
   Program8.FilmPrestretchFinalRev := 100;
   Program8.ArmSpeed := 100;
   Program8.CarriageDown4Top := 500;
   Program8.TopDownTime := 1500;
   Program8.LapsUnderTop := 0;
   Program8.Spare6 := 0;
   Program8.Spare7 := 0;
   Program8.Spare8 := 0;
   Program8.Spare9 := 0;
   Program8.Spare10 := 0;
   Program8.Spare11 := 0;
   Program8.Spare12 := 0;
   Program8.Overlap0_1 := 0;
   Program8.Height1 := 130;
   Program8.Landmark1 := FALSE;
   Program8.Lifter1 := FALSE;
   Program8.SpareBit1H1 := FALSE;
   Program8.Airblower1 := TRUE;
   Program8.NextStep1 := TRUE;
   Program8.PressureP1 := TRUE;
   Program8.SpareByte2H1 := 16#00;
   Program8.Revolution1 := 1;
   Program8.RopeUnit1_1 := 16#01;
   Program8.RopeUnit1_2 := 16#01;
   Program8.FilmForce1 := 5;
   Program8.FilmPrestretch1 := 200;
   Program8.Spare3H1 := 0;
   Program8.Spare49 := 0;
   Program8.Spare50 := 0;
   Program8.Spare51 := 0;
   Program8.Spare52 := 0;
   Program8.Spare53 := 0;
   Program8.Overlap1_2 := 0;
   Program8.Height2 := 50;
   Program8.Landmark2 := FALSE;
   Program8.Lifter2 := FALSE;
   Program8.SpareBit1H2 := FALSE;
   Program8.Airblower2 := TRUE;
   Program8.NextStep2 := TRUE;
   Program8.PressureP2 := TRUE;
   Program8.SpareByte2H2 := 16#00;
   Program8.Revolution2 := 1;
   Program8.RopeUnit2_1 := 16#01;
   Program8.RopeUnit2_2 := 16#01;
   Program8.FilmForce2 := 20;
   Program8.FilmPrestretch2 := 200;
   Program8.Spare3H2 := 0;
   Program8.Spare54 := 0;
   Program8.Spare55 := 0;
   Program8.Spare56 := 0;
   Program8.Spare57 := 0;
   Program8.Spare58 := 0;
   Program8.Overlap2_3 := 100;
   Program8.Height3 := -50;
   Program8.Landmark3 := TRUE;
   Program8.Lifter3 := FALSE;
   Program8.SpareBit1H3 := FALSE;
   Program8.Airblower3 := TRUE;
   Program8.NextStep3 := TRUE;
   Program8.PressureP3 := TRUE;
   Program8.SpareByte2H3 := 16#00;
   Program8.Revolution3 := 2;
   Program8.RopeUnit3_1 := 16#01;
   Program8.RopeUnit3_2 := 16#01;
   Program8.FilmForce3 := 30;
   Program8.FilmPrestretch3 := 200;
   Program8.Spare3H3 := 0;
   Program8.Spare59 := 0;
   Program8.Spare60 := 0;
   Program8.Spare61 := 380;
   Program8.Spare62 := 2800;
   Program8.Spare63 := 0;
   Program8.Overlap3_4 := 100;
   Program8.Height4 := 100;
   Program8.Landmark4 := FALSE;
   Program8.Lifter4 := FALSE;
   Program8.SpareBit1H4 := FALSE;
   Program8.Airblower4 := TRUE;
   Program8.NextStep4 := TRUE;
   Program8.PressureP4 := TRUE;
   Program8.SpareByte2H4 := 16#00;
   Program8.Revolution4 := 3;
   Program8.RopeUnit4_1 := 16#02;
   Program8.RopeUnit4_2 := 16#02;
   Program8.FilmForce4 := 30;
   Program8.FilmPrestretch4 := 200;
   Program8.Spare3H4 := 0;
   Program8.Spare64 := 0;
   Program8.Spare65 := 0;
   Program8.Spare66 := 0;
   Program8.Spare67 := 0;
   Program8.Spare68 := 0;
   Program8.Overlap4_5 := 0;
   Program8.Height5 := 50;
   Program8.Landmark5 := FALSE;
   Program8.Lifter5 := FALSE;
   Program8.SpareBit1H5 := FALSE;
   Program8.Airblower5 := TRUE;
   Program8.NextStep5 := FALSE;
   Program8.PressureP5 := FALSE;
   Program8.SpareByte2H5 := 16#00;
   Program8.Revolution5 := 1;
   Program8.RopeUnit5_1 := 16#01;
   Program8.RopeUnit5_2 := 16#01;
   Program8.FilmForce5 := 30;
   Program8.FilmPrestretch5 := 200;
   Program8.Spare3H5 := 0;
   Program8.Spare69 := 0;
   Program8.Spare70 := 0;
   Program8.Spare71 := 0;
   Program8.Spare72 := 0;
   Program8.Spare73 := 0;
   Program8.Overlap5_6 := 100;
   Program8.Height6 := 50;
   Program8.Landmark6 := FALSE;
   Program8.Lifter6 := FALSE;
   Program8.SpareBit1H6 := FALSE;
   Program8.Airblower6 := TRUE;
   Program8.NextStep6 := FALSE;
   Program8.PressureP6 := FALSE;
   Program8.SpareByte2H6 := 16#00;
   Program8.Revolution6 := 2;
   Program8.RopeUnit6_1 := 16#02;
   Program8.RopeUnit6_2 := 16#01;
   Program8.FilmForce6 := 20;
   Program8.FilmPrestretch6 := 200;
   Program8.Spare3H6 := 0;
   Program8.Spare74 := 0;
   Program8.Spare75 := 0;
   Program8.Spare76 := 0;
   Program8.Spare77 := 0;
   Program8.Spare78 := 0;
   Program8.Overlap6_7 := 0;
   Program8.Height7 := 0;
   Program8.Landmark7 := FALSE;
   Program8.Lifter7 := FALSE;
   Program8.SpareBit1H7 := FALSE;
   Program8.Airblower7 := FALSE;
   Program8.NextStep7 := TRUE;
   Program8.PressureP7 := FALSE;
   Program8.SpareByte2H7 := 16#00;
   Program8.Revolution7 := 1;
   Program8.RopeUnit7_1 := 16#01;
   Program8.RopeUnit7_2 := 16#01;
   Program8.FilmForce7 := 0;
   Program8.FilmPrestretch7 := 100;
   Program8.Spare3H7 := 0;
   Program8.Spare79 := 0;
   Program8.Spare80 := 0;
   Program8.Spare81 := 0;
   Program8.Spare82 := 0;
   Program8.Spare83 := 0;
   Program8.Overlap7_8 := 0;
   Program8.Height8 := 0;
   Program8.Landmark8 := FALSE;
   Program8.Lifter8 := FALSE;
   Program8.SpareBit1H8 := FALSE;
   Program8.Airblower8 := FALSE;
   Program8.NextStep8 := TRUE;
   Program8.PressureP8 := FALSE;
   Program8.SpareByte2H8 := 16#00;
   Program8.Revolution8 := 1;
   Program8.RopeUnit8_1 := 16#01;
   Program8.RopeUnit8_2 := 16#01;
   Program8.FilmForce8 := 0;
   Program8.FilmPrestretch8 := 100;
   Program8.Spare3H8 := 0;
   Program8.Spare84 := 0;
   Program8.Spare85 := 0;
   Program8.Spare86 := 0;
   Program8.Spare87 := 0;
   Program8.Spare88 := 0;
   Program8.Overlap8_9 := 0;
   Program8.Height9 := 0;
   Program8.Landmark9 := FALSE;
   Program8.Lifter9 := FALSE;
   Program8.SpareBit1H9 := FALSE;
   Program8.Airblower9 := FALSE;
   Program8.NextStep9 := TRUE;
   Program8.PressureP9 := FALSE;
   Program8.SpareByte2H9 := 16#00;
   Program8.Revolution9 := 1;
   Program8.RopeUnit9_1 := 16#01;
   Program8.RopeUnit9_2 := 16#01;
   Program8.FilmForce9 := 0;
   Program8.FilmPrestretch9 := 100;
   Program8.Spare3H9 := 0;
   Program8.Spare89 := 0;
   Program8.Spare90 := 0;
   Program8.Spare91 := 0;
   Program8.Spare92 := 0;
   Program8.Spare93 := 0;
   Program8.Overlap9_10 := 0;
   Program8.Height10 := 0;
   Program8.Landmark10 := FALSE;
   Program8.Lifter10 := FALSE;
   Program8.SpareBit1H10 := FALSE;
   Program8.Airblower10 := FALSE;
   Program8.NextStep10 := FALSE;
   Program8.PressureP10 := FALSE;
   Program8.SpareByte2H10 := 16#00;
   Program8.Revolution10 := 1;
   Program8.RopeUnit10_1 := 16#01;
   Program8.RopeUnit10_2 := 16#01;
   Program8.FilmForce10 := 0;
   Program8.FilmPrestretch10 := 100;
   Program8.Spare3H10 := 0;
   Program8.Spare94 := 0;
   Program8.Spare95 := 0;
   Program8.Spare96 := 0;
   Program8.Spare97 := 0;
   Program8.Spare98 := 0;
   Program8.Overlap10_11 := 0;
   Program8.Height11 := 0;
   Program8.Landmark11 := FALSE;
   Program8.Lifter11 := FALSE;
   Program8.SpareBit1H11 := FALSE;
   Program8.Airblower11 := FALSE;
   Program8.NextStep11 := TRUE;
   Program8.PressureP11 := FALSE;
   Program8.SpareByte2H11 := 16#00;
   Program8.Revolution11 := 1;
   Program8.RopeUnit11_1 := 16#01;
   Program8.RopeUnit11_2 := 16#01;
   Program8.FilmForce11 := 0;
   Program8.FilmPrestretch11 := 100;
   Program8.Spare3H11 := 0;
   Program8.Spare99 := 0;
   Program8.Spare100 := 0;
   Program8.Spare101 := 0;
   Program8.Spare102 := 0;
   Program8.Spare103 := 0;
   Program8.Overlap11_12 := 0;
   Program8.Height12 := 0;
   Program8.Landmark12 := FALSE;
   Program8.Lifter12 := FALSE;
   Program8.SpareBit1H12 := FALSE;
   Program8.Airblower12 := FALSE;
   Program8.NextStep12 := FALSE;
   Program8.PressureP12 := FALSE;
   Program8.SpareByte2H12 := 16#00;
   Program8.Revolution12 := 1;
   Program8.RopeUnit12_1 := 16#01;
   Program8.RopeUnit12_2 := 16#01;
   Program8.FilmForce12 := 0;
   Program8.FilmPrestretch12 := 100;
   Program8.Spare3H12 := 0;
   Program8.Spare104 := 0;
   Program8.Spare105 := 0;
   Program8.Spare106 := 0;
   Program8.Spare107 := 0;
   Program8.Spare108 := 0;
END_DATA_BLOCK

DATA_BLOCK "DB243_Program7"   // DB243
{ S7_Optimized_Access := 'FALSE' }
AUTHOR : Robopac
VERSION : 0.0
// stored: AutoNumber false, IsOnlyStoredInLoadMemory false, IsWriteProtectedInAS false
   VAR RETAIN
      Program7 { S7_SetPoint := 'True'} : "DatiProgramma";
   END_VAR
BEGIN
   Program7.Wrapping := TRUE;
   Program7.TopLenght := 500;
   Program7.TopRelease := 0;
   Program7.TopDown := 0;
   Program7.Top := 4;
   Program7.PressurePTime := 0;
   Program7.LifterTime := 0;
   Program7.RevOverContrast := 1;
   Program7.RopeEndCycle := 16#01;
   Program7.Spare4 := 16#01;
   Program7.RopeTime := 1500;
   Program7.RevOverClamp := 1;
   Program7.FilmForceFinalRev := 15;
   Program7.FilmPrestretchFinalRev := 100;
   Program7.ArmSpeed := 100;
   Program7.CarriageDown4Top := 500;
   Program7.TopDownTime := 1500;
   Program7.LapsUnderTop := 0;
   Program7.Spare6 := 0;
   Program7.Spare7 := 0;
   Program7.Spare8 := 0;
   Program7.Spare9 := 0;
   Program7.Spare10 := 0;
   Program7.Spare11 := 0;
   Program7.Spare12 := 0;
   Program7.Overlap0_1 := 0;
   Program7.Height1 := 15;
   Program7.Landmark1 := FALSE;
   Program7.Lifter1 := FALSE;
   Program7.SpareBit1H1 := FALSE;
   Program7.Airblower1 := TRUE;
   Program7.NextStep1 := TRUE;
   Program7.PressureP1 := TRUE;
   Program7.SpareByte2H1 := 16#00;
   Program7.Revolution1 := 0;
   Program7.RopeUnit1_1 := 16#02;
   Program7.RopeUnit1_2 := 16#01;
   Program7.FilmForce1 := 5;
   Program7.FilmPrestretch1 := 200;
   Program7.Spare3H1 := 0;
   Program7.Spare49 := 0;
   Program7.Spare50 := 0;
   Program7.Spare51 := 0;
   Program7.Spare52 := 0;
   Program7.Spare53 := 0;
   Program7.Overlap1_2 := 0;
   Program7.Height2 := 80;
   Program7.Landmark2 := FALSE;
   Program7.Lifter2 := FALSE;
   Program7.SpareBit1H2 := FALSE;
   Program7.Airblower2 := TRUE;
   Program7.NextStep2 := TRUE;
   Program7.PressureP2 := TRUE;
   Program7.SpareByte2H2 := 16#00;
   Program7.Revolution2 := 1;
   Program7.RopeUnit2_1 := 16#01;
   Program7.RopeUnit2_2 := 16#01;
   Program7.FilmForce2 := 15;
   Program7.FilmPrestretch2 := 200;
   Program7.Spare3H2 := 0;
   Program7.Spare54 := 0;
   Program7.Spare55 := 0;
   Program7.Spare56 := 0;
   Program7.Spare57 := 0;
   Program7.Spare58 := 0;
   Program7.Overlap2_3 := 0;
   Program7.Height3 := 120;
   Program7.Landmark3 := FALSE;
   Program7.Lifter3 := FALSE;
   Program7.SpareBit1H3 := FALSE;
   Program7.Airblower3 := TRUE;
   Program7.NextStep3 := TRUE;
   Program7.PressureP3 := TRUE;
   Program7.SpareByte2H3 := 16#00;
   Program7.Revolution3 := 1;
   Program7.RopeUnit3_1 := 16#01;
   Program7.RopeUnit3_2 := 16#01;
   Program7.FilmForce3 := 25;
   Program7.FilmPrestretch3 := 200;
   Program7.Spare3H3 := 0;
   Program7.Spare59 := 0;
   Program7.Spare60 := 0;
   Program7.Spare61 := 380;
   Program7.Spare62 := 2800;
   Program7.Spare63 := 0;
   Program7.Overlap3_4 := 0;
   Program7.Height4 := -100;
   Program7.Landmark4 := TRUE;
   Program7.Lifter4 := FALSE;
   Program7.SpareBit1H4 := FALSE;
   Program7.Airblower4 := FALSE;
   Program7.NextStep4 := TRUE;
   Program7.PressureP4 := TRUE;
   Program7.SpareByte2H4 := 16#00;
   Program7.Revolution4 := 1;
   Program7.RopeUnit4_1 := 16#01;
   Program7.RopeUnit4_2 := 16#01;
   Program7.FilmForce4 := 20;
   Program7.FilmPrestretch4 := 200;
   Program7.Spare3H4 := 0;
   Program7.Spare64 := 0;
   Program7.Spare65 := 0;
   Program7.Spare66 := 0;
   Program7.Spare67 := 0;
   Program7.Spare68 := 0;
   Program7.Overlap4_5 := 300;
   Program7.Height5 := 120;
   Program7.Landmark5 := FALSE;
   Program7.Lifter5 := FALSE;
   Program7.SpareBit1H5 := FALSE;
   Program7.Airblower5 := TRUE;
   Program7.NextStep5 := TRUE;
   Program7.PressureP5 := FALSE;
   Program7.SpareByte2H5 := 16#00;
   Program7.Revolution5 := 2;
   Program7.RopeUnit5_1 := 16#02;
   Program7.RopeUnit5_2 := 16#02;
   Program7.FilmForce5 := 15;
   Program7.FilmPrestretch5 := 200;
   Program7.Spare3H5 := 0;
   Program7.Spare69 := 0;
   Program7.Spare70 := 0;
   Program7.Spare71 := 0;
   Program7.Spare72 := 0;
   Program7.Spare73 := 0;
   Program7.Overlap5_6 := 300;
   Program7.Height6 := 85;
   Program7.Landmark6 := FALSE;
   Program7.Lifter6 := FALSE;
   Program7.SpareBit1H6 := FALSE;
   Program7.Airblower6 := TRUE;
   Program7.NextStep6 := FALSE;
   Program7.PressureP6 := FALSE;
   Program7.SpareByte2H6 := 16#00;
   Program7.Revolution6 := 1;
   Program7.RopeUnit6_1 := 16#01;
   Program7.RopeUnit6_2 := 16#01;
   Program7.FilmForce6 := 20;
   Program7.FilmPrestretch6 := 200;
   Program7.Spare3H6 := 0;
   Program7.Spare74 := 0;
   Program7.Spare75 := 0;
   Program7.Spare76 := 0;
   Program7.Spare77 := 0;
   Program7.Spare78 := 0;
   Program7.Overlap6_7 := 0;
   Program7.Height7 := 0;
   Program7.Landmark7 := FALSE;
   Program7.Lifter7 := FALSE;
   Program7.SpareBit1H7 := FALSE;
   Program7.Airblower7 := FALSE;
   Program7.NextStep7 := TRUE;
   Program7.PressureP7 := FALSE;
   Program7.SpareByte2H7 := 16#00;
   Program7.Revolution7 := 1;
   Program7.RopeUnit7_1 := 16#01;
   Program7.RopeUnit7_2 := 16#01;
   Program7.FilmForce7 := 0;
   Program7.FilmPrestretch7 := 100;
   Program7.Spare3H7 := 0;
   Program7.Spare79 := 0;
   Program7.Spare80 := 0;
   Program7.Spare81 := 0;
   Program7.Spare82 := 0;
   Program7.Spare83 := 0;
   Program7.Overlap7_8 := 0;
   Program7.Height8 := 0;
   Program7.Landmark8 := FALSE;
   Program7.Lifter8 := FALSE;
   Program7.SpareBit1H8 := FALSE;
   Program7.Airblower8 := FALSE;
   Program7.NextStep8 := TRUE;
   Program7.PressureP8 := FALSE;
   Program7.SpareByte2H8 := 16#00;
   Program7.Revolution8 := 1;
   Program7.RopeUnit8_1 := 16#01;
   Program7.RopeUnit8_2 := 16#01;
   Program7.FilmForce8 := 0;
   Program7.FilmPrestretch8 := 100;
   Program7.Spare3H8 := 0;
   Program7.Spare84 := 0;
   Program7.Spare85 := 0;
   Program7.Spare86 := 0;
   Program7.Spare87 := 0;
   Program7.Spare88 := 0;
   Program7.Overlap8_9 := 0;
   Program7.Height9 := 0;
   Program7.Landmark9 := FALSE;
   Program7.Lifter9 := FALSE;
   Program7.SpareBit1H9 := FALSE;
   Program7.Airblower9 := FALSE;
   Program7.NextStep9 := TRUE;
   Program7.PressureP9 := FALSE;
   Program7.SpareByte2H9 := 16#00;
   Program7.Revolution9 := 1;
   Program7.RopeUnit9_1 := 16#01;
   Program7.RopeUnit9_2 := 16#01;
   Program7.FilmForce9 := 0;
   Program7.FilmPrestretch9 := 100;
   Program7.Spare3H9 := 0;
   Program7.Spare89 := 0;
   Program7.Spare90 := 0;
   Program7.Spare91 := 0;
   Program7.Spare92 := 0;
   Program7.Spare93 := 0;
   Program7.Overlap9_10 := 0;
   Program7.Height10 := 0;
   Program7.Landmark10 := FALSE;
   Program7.Lifter10 := FALSE;
   Program7.SpareBit1H10 := FALSE;
   Program7.Airblower10 := FALSE;
   Program7.NextStep10 := FALSE;
   Program7.PressureP10 := FALSE;
   Program7.SpareByte2H10 := 16#00;
   Program7.Revolution10 := 1;
   Program7.RopeUnit10_1 := 16#01;
   Program7.RopeUnit10_2 := 16#01;
   Program7.FilmForce10 := 0;
   Program7.FilmPrestretch10 := 100;
   Program7.Spare3H10 := 0;
   Program7.Spare94 := 0;
   Program7.Spare95 := 0;
   Program7.Spare96 := 0;
   Program7.Spare97 := 0;
   Program7.Spare98 := 0;
   Program7.Overlap10_11 := 0;
   Program7.Height11 := 0;
   Program7.Landmark11 := FALSE;
   Program7.Lifter11 := FALSE;
   Program7.SpareBit1H11 := FALSE;
   Program7.Airblower11 := FALSE;
   Program7.NextStep11 := TRUE;
   Program7.PressureP11 := FALSE;
   Program7.SpareByte2H11 := 16#00;
   Program7.Revolution11 := 1;
   Program7.RopeUnit11_1 := 16#01;
   Program7.RopeUnit11_2 := 16#01;
   Program7.FilmForce11 := 0;
   Program7.FilmPrestretch11 := 100;
   Program7.Spare3H11 := 0;
   Program7.Spare99 := 0;
   Program7.Spare100 := 0;
   Program7.Spare101 := 0;
   Program7.Spare102 := 0;
   Program7.Spare103 := 0;
   Program7.Overlap11_12 := 0;
   Program7.Height12 := 0;
   Program7.Landmark12 := FALSE;
   Program7.Lifter12 := FALSE;
   Program7.SpareBit1H12 := FALSE;
   Program7.Airblower12 := FALSE;
   Program7.NextStep12 := FALSE;
   Program7.PressureP12 := FALSE;
   Program7.SpareByte2H12 := 16#00;
   Program7.Revolution12 := 1;
   Program7.RopeUnit12_1 := 16#01;
   Program7.RopeUnit12_2 := 16#01;
   Program7.FilmForce12 := 0;
   Program7.FilmPrestretch12 := 100;
   Program7.Spare3H12 := 0;
   Program7.Spare104 := 0;
   Program7.Spare105 := 0;
   Program7.Spare106 := 0;
   Program7.Spare107 := 0;
   Program7.Spare108 := 0;
END_DATA_BLOCK

DATA_BLOCK "DB244_Program6"   // DB244
{ S7_Optimized_Access := 'FALSE' }
AUTHOR : Robopac
VERSION : 0.0
// stored: AutoNumber false, IsOnlyStoredInLoadMemory false, IsWriteProtectedInAS false
   VAR RETAIN
      Program6 { S7_SetPoint := 'True'} : "DatiProgramma";
   END_VAR
BEGIN
   Program6.Wrapping := TRUE;
   Program6.TopLenght := 500;
   Program6.TopRelease := 0;
   Program6.TopDown := 0;
   Program6.Top := 4;
   Program6.PressurePTime := 0;
   Program6.LifterTime := 0;
   Program6.RevOverContrast := 1;
   Program6.RopeEndCycle := 16#02;
   Program6.Spare4 := 16#01;
   Program6.RopeTime := 1500;
   Program6.RevOverClamp := 1;
   Program6.FilmForceFinalRev := 10;
   Program6.FilmPrestretchFinalRev := 100;
   Program6.ArmSpeed := 100;
   Program6.CarriageDown4Top := 500;
   Program6.TopDownTime := 1500;
   Program6.LapsUnderTop := 0;
   Program6.Spare6 := 0;
   Program6.Spare7 := 0;
   Program6.Spare8 := 0;
   Program6.Spare9 := 0;
   Program6.Spare10 := 0;
   Program6.Spare11 := 0;
   Program6.Spare12 := 0;
   Program6.Overlap0_1 := 0;
   Program6.Height1 := 130;
   Program6.Landmark1 := FALSE;
   Program6.Lifter1 := FALSE;
   Program6.SpareBit1H1 := FALSE;
   Program6.Airblower1 := TRUE;
   Program6.NextStep1 := TRUE;
   Program6.PressureP1 := TRUE;
   Program6.SpareByte2H1 := 16#00;
   Program6.Revolution1 := 1;
   Program6.RopeUnit1_1 := 16#01;
   Program6.RopeUnit1_2 := 16#01;
   Program6.FilmForce1 := 5;
   Program6.FilmPrestretch1 := 200;
   Program6.Spare3H1 := 0;
   Program6.Spare49 := 0;
   Program6.Spare50 := 0;
   Program6.Spare51 := 0;
   Program6.Spare52 := 0;
   Program6.Spare53 := 0;
   Program6.Overlap1_2 := 0;
   Program6.Height2 := 50;
   Program6.Landmark2 := FALSE;
   Program6.Lifter2 := FALSE;
   Program6.SpareBit1H2 := FALSE;
   Program6.Airblower2 := TRUE;
   Program6.NextStep2 := TRUE;
   Program6.PressureP2 := TRUE;
   Program6.SpareByte2H2 := 16#00;
   Program6.Revolution2 := 1;
   Program6.RopeUnit2_1 := 16#01;
   Program6.RopeUnit2_2 := 16#01;
   Program6.FilmForce2 := 20;
   Program6.FilmPrestretch2 := 200;
   Program6.Spare3H2 := 0;
   Program6.Spare54 := 0;
   Program6.Spare55 := 0;
   Program6.Spare56 := 0;
   Program6.Spare57 := 0;
   Program6.Spare58 := 0;
   Program6.Overlap2_3 := 100;
   Program6.Height3 := -50;
   Program6.Landmark3 := TRUE;
   Program6.Lifter3 := FALSE;
   Program6.SpareBit1H3 := FALSE;
   Program6.Airblower3 := TRUE;
   Program6.NextStep3 := TRUE;
   Program6.PressureP3 := TRUE;
   Program6.SpareByte2H3 := 16#00;
   Program6.Revolution3 := 2;
   Program6.RopeUnit3_1 := 16#01;
   Program6.RopeUnit3_2 := 16#01;
   Program6.FilmForce3 := 30;
   Program6.FilmPrestretch3 := 200;
   Program6.Spare3H3 := 0;
   Program6.Spare59 := 0;
   Program6.Spare60 := 0;
   Program6.Spare61 := 380;
   Program6.Spare62 := 2800;
   Program6.Spare63 := 0;
   Program6.Overlap3_4 := 100;
   Program6.Height4 := 100;
   Program6.Landmark4 := FALSE;
   Program6.Lifter4 := FALSE;
   Program6.SpareBit1H4 := FALSE;
   Program6.Airblower4 := TRUE;
   Program6.NextStep4 := TRUE;
   Program6.PressureP4 := TRUE;
   Program6.SpareByte2H4 := 16#00;
   Program6.Revolution4 := 3;
   Program6.RopeUnit4_1 := 16#02;
   Program6.RopeUnit4_2 := 16#02;
   Program6.FilmForce4 := 30;
   Program6.FilmPrestretch4 := 200;
   Program6.Spare3H4 := 0;
   Program6.Spare64 := 0;
   Program6.Spare65 := 0;
   Program6.Spare66 := 0;
   Program6.Spare67 := 0;
   Program6.Spare68 := 0;
   Program6.Overlap4_5 := 0;
   Program6.Height5 := 50;
   Program6.Landmark5 := FALSE;
   Program6.Lifter5 := FALSE;
   Program6.SpareBit1H5 := FALSE;
   Program6.Airblower5 := TRUE;
   Program6.NextStep5 := FALSE;
   Program6.PressureP5 := FALSE;
   Program6.SpareByte2H5 := 16#00;
   Program6.Revolution5 := 1;
   Program6.RopeUnit5_1 := 16#01;
   Program6.RopeUnit5_2 := 16#01;
   Program6.FilmForce5 := 30;
   Program6.FilmPrestretch5 := 200;
   Program6.Spare3H5 := 0;
   Program6.Spare69 := 0;
   Program6.Spare70 := 0;
   Program6.Spare71 := 0;
   Program6.Spare72 := 0;
   Program6.Spare73 := 0;
   Program6.Overlap5_6 := 100;
   Program6.Height6 := 50;
   Program6.Landmark6 := FALSE;
   Program6.Lifter6 := FALSE;
   Program6.SpareBit1H6 := FALSE;
   Program6.Airblower6 := TRUE;
   Program6.NextStep6 := FALSE;
   Program6.PressureP6 := FALSE;
   Program6.SpareByte2H6 := 16#00;
   Program6.Revolution6 := 2;
   Program6.RopeUnit6_1 := 16#02;
   Program6.RopeUnit6_2 := 16#01;
   Program6.FilmForce6 := 20;
   Program6.FilmPrestretch6 := 200;
   Program6.Spare3H6 := 0;
   Program6.Spare74 := 0;
   Program6.Spare75 := 0;
   Program6.Spare76 := 0;
   Program6.Spare77 := 0;
   Program6.Spare78 := 0;
   Program6.Overlap6_7 := 0;
   Program6.Height7 := 0;
   Program6.Landmark7 := FALSE;
   Program6.Lifter7 := FALSE;
   Program6.SpareBit1H7 := FALSE;
   Program6.Airblower7 := FALSE;
   Program6.NextStep7 := TRUE;
   Program6.PressureP7 := FALSE;
   Program6.SpareByte2H7 := 16#00;
   Program6.Revolution7 := 1;
   Program6.RopeUnit7_1 := 16#01;
   Program6.RopeUnit7_2 := 16#01;
   Program6.FilmForce7 := 0;
   Program6.FilmPrestretch7 := 100;
   Program6.Spare3H7 := 0;
   Program6.Spare79 := 0;
   Program6.Spare80 := 0;
   Program6.Spare81 := 0;
   Program6.Spare82 := 0;
   Program6.Spare83 := 0;
   Program6.Overlap7_8 := 0;
   Program6.Height8 := 0;
   Program6.Landmark8 := FALSE;
   Program6.Lifter8 := FALSE;
   Program6.SpareBit1H8 := FALSE;
   Program6.Airblower8 := FALSE;
   Program6.NextStep8 := TRUE;
   Program6.PressureP8 := FALSE;
   Program6.SpareByte2H8 := 16#00;
   Program6.Revolution8 := 1;
   Program6.RopeUnit8_1 := 16#01;
   Program6.RopeUnit8_2 := 16#01;
   Program6.FilmForce8 := 0;
   Program6.FilmPrestretch8 := 100;
   Program6.Spare3H8 := 0;
   Program6.Spare84 := 0;
   Program6.Spare85 := 0;
   Program6.Spare86 := 0;
   Program6.Spare87 := 0;
   Program6.Spare88 := 0;
   Program6.Overlap8_9 := 0;
   Program6.Height9 := 0;
   Program6.Landmark9 := FALSE;
   Program6.Lifter9 := FALSE;
   Program6.SpareBit1H9 := FALSE;
   Program6.Airblower9 := FALSE;
   Program6.NextStep9 := TRUE;
   Program6.PressureP9 := FALSE;
   Program6.SpareByte2H9 := 16#00;
   Program6.Revolution9 := 1;
   Program6.RopeUnit9_1 := 16#01;
   Program6.RopeUnit9_2 := 16#01;
   Program6.FilmForce9 := 0;
   Program6.FilmPrestretch9 := 100;
   Program6.Spare3H9 := 0;
   Program6.Spare89 := 0;
   Program6.Spare90 := 0;
   Program6.Spare91 := 0;
   Program6.Spare92 := 0;
   Program6.Spare93 := 0;
   Program6.Overlap9_10 := 0;
   Program6.Height10 := 0;
   Program6.Landmark10 := FALSE;
   Program6.Lifter10 := FALSE;
   Program6.SpareBit1H10 := FALSE;
   Program6.Airblower10 := FALSE;
   Program6.NextStep10 := FALSE;
   Program6.PressureP10 := FALSE;
   Program6.SpareByte2H10 := 16#00;
   Program6.Revolution10 := 1;
   Program6.RopeUnit10_1 := 16#01;
   Program6.RopeUnit10_2 := 16#01;
   Program6.FilmForce10 := 0;
   Program6.FilmPrestretch10 := 100;
   Program6.Spare3H10 := 0;
   Program6.Spare94 := 0;
   Program6.Spare95 := 0;
   Program6.Spare96 := 0;
   Program6.Spare97 := 0;
   Program6.Spare98 := 0;
   Program6.Overlap10_11 := 0;
   Program6.Height11 := 0;
   Program6.Landmark11 := FALSE;
   Program6.Lifter11 := FALSE;
   Program6.SpareBit1H11 := FALSE;
   Program6.Airblower11 := FALSE;
   Program6.NextStep11 := TRUE;
   Program6.PressureP11 := FALSE;
   Program6.SpareByte2H11 := 16#00;
   Program6.Revolution11 := 1;
   Program6.RopeUnit11_1 := 16#01;
   Program6.RopeUnit11_2 := 16#01;
   Program6.FilmForce11 := 0;
   Program6.FilmPrestretch11 := 100;
   Program6.Spare3H11 := 0;
   Program6.Spare99 := 0;
   Program6.Spare100 := 0;
   Program6.Spare101 := 0;
   Program6.Spare102 := 0;
   Program6.Spare103 := 0;
   Program6.Overlap11_12 := 0;
   Program6.Height12 := 0;
   Program6.Landmark12 := FALSE;
   Program6.Lifter12 := FALSE;
   Program6.SpareBit1H12 := FALSE;
   Program6.Airblower12 := FALSE;
   Program6.NextStep12 := FALSE;
   Program6.PressureP12 := FALSE;
   Program6.SpareByte2H12 := 16#00;
   Program6.Revolution12 := 1;
   Program6.RopeUnit12_1 := 16#01;
   Program6.RopeUnit12_2 := 16#01;
   Program6.FilmForce12 := 0;
   Program6.FilmPrestretch12 := 100;
   Program6.Spare3H12 := 0;
   Program6.Spare104 := 0;
   Program6.Spare105 := 0;
   Program6.Spare106 := 0;
   Program6.Spare107 := 0;
   Program6.Spare108 := 0;
END_DATA_BLOCK

DATA_BLOCK "DB245_Program5"   // DB245
{ S7_Optimized_Access := 'FALSE' }
AUTHOR : Robopac
VERSION : 0.0
// stored: AutoNumber false, IsOnlyStoredInLoadMemory false, IsWriteProtectedInAS false
   VAR RETAIN
      Program5 { S7_SetPoint := 'True'} : "DatiProgramma";
   END_VAR
BEGIN
   Program5.Wrapping := TRUE;
   Program5.TopLenght := 500;
   Program5.TopRelease := 0;
   Program5.TopDown := 0;
   Program5.Top := 4;
   Program5.PressurePTime := 0;
   Program5.LifterTime := 0;
   Program5.RevOverContrast := 1;
   Program5.RopeEndCycle := 16#02;
   Program5.Spare4 := 16#01;
   Program5.RopeTime := 1500;
   Program5.RevOverClamp := 1;
   Program5.FilmForceFinalRev := 10;
   Program5.FilmPrestretchFinalRev := 100;
   Program5.ArmSpeed := 100;
   Program5.CarriageDown4Top := 500;
   Program5.TopDownTime := 1500;
   Program5.LapsUnderTop := 0;
   Program5.Spare6 := 0;
   Program5.Spare7 := 0;
   Program5.Spare8 := 0;
   Program5.Spare9 := 0;
   Program5.Spare10 := 0;
   Program5.Spare11 := 0;
   Program5.Spare12 := 0;
   Program5.Overlap0_1 := 0;
   Program5.Height1 := 130;
   Program5.Landmark1 := FALSE;
   Program5.Lifter1 := FALSE;
   Program5.SpareBit1H1 := FALSE;
   Program5.Airblower1 := TRUE;
   Program5.NextStep1 := TRUE;
   Program5.PressureP1 := TRUE;
   Program5.SpareByte2H1 := 16#00;
   Program5.Revolution1 := 1;
   Program5.RopeUnit1_1 := 16#01;
   Program5.RopeUnit1_2 := 16#01;
   Program5.FilmForce1 := 5;
   Program5.FilmPrestretch1 := 200;
   Program5.Spare3H1 := 0;
   Program5.Spare49 := 0;
   Program5.Spare50 := 0;
   Program5.Spare51 := 0;
   Program5.Spare52 := 0;
   Program5.Spare53 := 0;
   Program5.Overlap1_2 := 0;
   Program5.Height2 := 50;
   Program5.Landmark2 := FALSE;
   Program5.Lifter2 := FALSE;
   Program5.SpareBit1H2 := FALSE;
   Program5.Airblower2 := TRUE;
   Program5.NextStep2 := TRUE;
   Program5.PressureP2 := TRUE;
   Program5.SpareByte2H2 := 16#00;
   Program5.Revolution2 := 1;
   Program5.RopeUnit2_1 := 16#01;
   Program5.RopeUnit2_2 := 16#01;
   Program5.FilmForce2 := 20;
   Program5.FilmPrestretch2 := 200;
   Program5.Spare3H2 := 0;
   Program5.Spare54 := 0;
   Program5.Spare55 := 0;
   Program5.Spare56 := 0;
   Program5.Spare57 := 0;
   Program5.Spare58 := 0;
   Program5.Overlap2_3 := 100;
   Program5.Height3 := -50;
   Program5.Landmark3 := TRUE;
   Program5.Lifter3 := FALSE;
   Program5.SpareBit1H3 := FALSE;
   Program5.Airblower3 := TRUE;
   Program5.NextStep3 := TRUE;
   Program5.PressureP3 := TRUE;
   Program5.SpareByte2H3 := 16#00;
   Program5.Revolution3 := 2;
   Program5.RopeUnit3_1 := 16#01;
   Program5.RopeUnit3_2 := 16#01;
   Program5.FilmForce3 := 30;
   Program5.FilmPrestretch3 := 200;
   Program5.Spare3H3 := 0;
   Program5.Spare59 := 0;
   Program5.Spare60 := 0;
   Program5.Spare61 := 380;
   Program5.Spare62 := 2800;
   Program5.Spare63 := 0;
   Program5.Overlap3_4 := 100;
   Program5.Height4 := 100;
   Program5.Landmark4 := FALSE;
   Program5.Lifter4 := FALSE;
   Program5.SpareBit1H4 := FALSE;
   Program5.Airblower4 := TRUE;
   Program5.NextStep4 := TRUE;
   Program5.PressureP4 := TRUE;
   Program5.SpareByte2H4 := 16#00;
   Program5.Revolution4 := 3;
   Program5.RopeUnit4_1 := 16#02;
   Program5.RopeUnit4_2 := 16#02;
   Program5.FilmForce4 := 30;
   Program5.FilmPrestretch4 := 200;
   Program5.Spare3H4 := 0;
   Program5.Spare64 := 0;
   Program5.Spare65 := 0;
   Program5.Spare66 := 0;
   Program5.Spare67 := 0;
   Program5.Spare68 := 0;
   Program5.Overlap4_5 := 0;
   Program5.Height5 := 50;
   Program5.Landmark5 := FALSE;
   Program5.Lifter5 := FALSE;
   Program5.SpareBit1H5 := FALSE;
   Program5.Airblower5 := TRUE;
   Program5.NextStep5 := FALSE;
   Program5.PressureP5 := FALSE;
   Program5.SpareByte2H5 := 16#00;
   Program5.Revolution5 := 1;
   Program5.RopeUnit5_1 := 16#01;
   Program5.RopeUnit5_2 := 16#01;
   Program5.FilmForce5 := 30;
   Program5.FilmPrestretch5 := 200;
   Program5.Spare3H5 := 0;
   Program5.Spare69 := 0;
   Program5.Spare70 := 0;
   Program5.Spare71 := 0;
   Program5.Spare72 := 0;
   Program5.Spare73 := 0;
   Program5.Overlap5_6 := 100;
   Program5.Height6 := 50;
   Program5.Landmark6 := FALSE;
   Program5.Lifter6 := FALSE;
   Program5.SpareBit1H6 := FALSE;
   Program5.Airblower6 := TRUE;
   Program5.NextStep6 := FALSE;
   Program5.PressureP6 := FALSE;
   Program5.SpareByte2H6 := 16#00;
   Program5.Revolution6 := 2;
   Program5.RopeUnit6_1 := 16#02;
   Program5.RopeUnit6_2 := 16#01;
   Program5.FilmForce6 := 20;
   Program5.FilmPrestretch6 := 200;
   Program5.Spare3H6 := 0;
   Program5.Spare74 := 0;
   Program5.Spare75 := 0;
   Program5.Spare76 := 0;
   Program5.Spare77 := 0;
   Program5.Spare78 := 0;
   Program5.Overlap6_7 := 0;
   Program5.Height7 := 0;
   Program5.Landmark7 := FALSE;
   Program5.Lifter7 := FALSE;
   Program5.SpareBit1H7 := FALSE;
   Program5.Airblower7 := FALSE;
   Program5.NextStep7 := TRUE;
   Program5.PressureP7 := FALSE;
   Program5.SpareByte2H7 := 16#00;
   Program5.Revolution7 := 1;
   Program5.RopeUnit7_1 := 16#01;
   Program5.RopeUnit7_2 := 16#01;
   Program5.FilmForce7 := 0;
   Program5.FilmPrestretch7 := 100;
   Program5.Spare3H7 := 0;
   Program5.Spare79 := 0;
   Program5.Spare80 := 0;
   Program5.Spare81 := 0;
   Program5.Spare82 := 0;
   Program5.Spare83 := 0;
   Program5.Overlap7_8 := 0;
   Program5.Height8 := 0;
   Program5.Landmark8 := FALSE;
   Program5.Lifter8 := FALSE;
   Program5.SpareBit1H8 := FALSE;
   Program5.Airblower8 := FALSE;
   Program5.NextStep8 := TRUE;
   Program5.PressureP8 := FALSE;
   Program5.SpareByte2H8 := 16#00;
   Program5.Revolution8 := 1;
   Program5.RopeUnit8_1 := 16#01;
   Program5.RopeUnit8_2 := 16#01;
   Program5.FilmForce8 := 0;
   Program5.FilmPrestretch8 := 100;
   Program5.Spare3H8 := 0;
   Program5.Spare84 := 0;
   Program5.Spare85 := 0;
   Program5.Spare86 := 0;
   Program5.Spare87 := 0;
   Program5.Spare88 := 0;
   Program5.Overlap8_9 := 0;
   Program5.Height9 := 0;
   Program5.Landmark9 := FALSE;
   Program5.Lifter9 := FALSE;
   Program5.SpareBit1H9 := FALSE;
   Program5.Airblower9 := FALSE;
   Program5.NextStep9 := TRUE;
   Program5.PressureP9 := FALSE;
   Program5.SpareByte2H9 := 16#00;
   Program5.Revolution9 := 1;
   Program5.RopeUnit9_1 := 16#01;
   Program5.RopeUnit9_2 := 16#01;
   Program5.FilmForce9 := 0;
   Program5.FilmPrestretch9 := 100;
   Program5.Spare3H9 := 0;
   Program5.Spare89 := 0;
   Program5.Spare90 := 0;
   Program5.Spare91 := 0;
   Program5.Spare92 := 0;
   Program5.Spare93 := 0;
   Program5.Overlap9_10 := 0;
   Program5.Height10 := 0;
   Program5.Landmark10 := FALSE;
   Program5.Lifter10 := FALSE;
   Program5.SpareBit1H10 := FALSE;
   Program5.Airblower10 := FALSE;
   Program5.NextStep10 := FALSE;
   Program5.PressureP10 := FALSE;
   Program5.SpareByte2H10 := 16#00;
   Program5.Revolution10 := 1;
   Program5.RopeUnit10_1 := 16#01;
   Program5.RopeUnit10_2 := 16#01;
   Program5.FilmForce10 := 0;
   Program5.FilmPrestretch10 := 100;
   Program5.Spare3H10 := 0;
   Program5.Spare94 := 0;
   Program5.Spare95 := 0;
   Program5.Spare96 := 0;
   Program5.Spare97 := 0;
   Program5.Spare98 := 0;
   Program5.Overlap10_11 := 0;
   Program5.Height11 := 0;
   Program5.Landmark11 := FALSE;
   Program5.Lifter11 := FALSE;
   Program5.SpareBit1H11 := FALSE;
   Program5.Airblower11 := FALSE;
   Program5.NextStep11 := TRUE;
   Program5.PressureP11 := FALSE;
   Program5.SpareByte2H11 := 16#00;
   Program5.Revolution11 := 1;
   Program5.RopeUnit11_1 := 16#01;
   Program5.RopeUnit11_2 := 16#01;
   Program5.FilmForce11 := 0;
   Program5.FilmPrestretch11 := 100;
   Program5.Spare3H11 := 0;
   Program5.Spare99 := 0;
   Program5.Spare100 := 0;
   Program5.Spare101 := 0;
   Program5.Spare102 := 0;
   Program5.Spare103 := 0;
   Program5.Overlap11_12 := 0;
   Program5.Height12 := 0;
   Program5.Landmark12 := FALSE;
   Program5.Lifter12 := FALSE;
   Program5.SpareBit1H12 := FALSE;
   Program5.Airblower12 := FALSE;
   Program5.NextStep12 := FALSE;
   Program5.PressureP12 := FALSE;
   Program5.SpareByte2H12 := 16#00;
   Program5.Revolution12 := 1;
   Program5.RopeUnit12_1 := 16#01;
   Program5.RopeUnit12_2 := 16#01;
   Program5.FilmForce12 := 0;
   Program5.FilmPrestretch12 := 100;
   Program5.Spare3H12 := 0;
   Program5.Spare104 := 0;
   Program5.Spare105 := 0;
   Program5.Spare106 := 0;
   Program5.Spare107 := 0;
   Program5.Spare108 := 0;
END_DATA_BLOCK

DATA_BLOCK "DB246_Program4"   // DB246
{ S7_Optimized_Access := 'FALSE' }
AUTHOR : Robopac
VERSION : 0.0
// stored: AutoNumber false, IsOnlyStoredInLoadMemory false, IsWriteProtectedInAS false
   VAR RETAIN
      Program4 { S7_SetPoint := 'True'} : "DatiProgramma";
   END_VAR
BEGIN
   Program4.Wrapping := TRUE;
   Program4.TopLenght := 500;
   Program4.TopRelease := 0;
   Program4.TopDown := 0;
   Program4.Top := 4;
   Program4.PressurePTime := 0;
   Program4.LifterTime := 0;
   Program4.RevOverContrast := 1;
   Program4.RopeEndCycle := 16#02;
   Program4.Spare4 := 16#01;
   Program4.RopeTime := 1500;
   Program4.RevOverClamp := 1;
   Program4.FilmForceFinalRev := 10;
   Program4.FilmPrestretchFinalRev := 100;
   Program4.ArmSpeed := 100;
   Program4.CarriageDown4Top := 500;
   Program4.TopDownTime := 1500;
   Program4.LapsUnderTop := 0;
   Program4.Spare6 := 0;
   Program4.Spare7 := 0;
   Program4.Spare8 := 0;
   Program4.Spare9 := 0;
   Program4.Spare10 := 0;
   Program4.Spare11 := 0;
   Program4.Spare12 := 0;
   Program4.Overlap0_1 := 0;
   Program4.Height1 := 130;
   Program4.Landmark1 := FALSE;
   Program4.Lifter1 := FALSE;
   Program4.SpareBit1H1 := FALSE;
   Program4.Airblower1 := TRUE;
   Program4.NextStep1 := TRUE;
   Program4.PressureP1 := TRUE;
   Program4.SpareByte2H1 := 16#00;
   Program4.Revolution1 := 1;
   Program4.RopeUnit1_1 := 16#01;
   Program4.RopeUnit1_2 := 16#01;
   Program4.FilmForce1 := 5;
   Program4.FilmPrestretch1 := 200;
   Program4.Spare3H1 := 0;
   Program4.Spare49 := 0;
   Program4.Spare50 := 0;
   Program4.Spare51 := 0;
   Program4.Spare52 := 0;
   Program4.Spare53 := 0;
   Program4.Overlap1_2 := 0;
   Program4.Height2 := 50;
   Program4.Landmark2 := FALSE;
   Program4.Lifter2 := FALSE;
   Program4.SpareBit1H2 := FALSE;
   Program4.Airblower2 := TRUE;
   Program4.NextStep2 := TRUE;
   Program4.PressureP2 := TRUE;
   Program4.SpareByte2H2 := 16#00;
   Program4.Revolution2 := 1;
   Program4.RopeUnit2_1 := 16#01;
   Program4.RopeUnit2_2 := 16#01;
   Program4.FilmForce2 := 20;
   Program4.FilmPrestretch2 := 200;
   Program4.Spare3H2 := 0;
   Program4.Spare54 := 0;
   Program4.Spare55 := 0;
   Program4.Spare56 := 0;
   Program4.Spare57 := 0;
   Program4.Spare58 := 0;
   Program4.Overlap2_3 := 100;
   Program4.Height3 := -50;
   Program4.Landmark3 := TRUE;
   Program4.Lifter3 := FALSE;
   Program4.SpareBit1H3 := FALSE;
   Program4.Airblower3 := TRUE;
   Program4.NextStep3 := TRUE;
   Program4.PressureP3 := TRUE;
   Program4.SpareByte2H3 := 16#00;
   Program4.Revolution3 := 2;
   Program4.RopeUnit3_1 := 16#01;
   Program4.RopeUnit3_2 := 16#01;
   Program4.FilmForce3 := 30;
   Program4.FilmPrestretch3 := 200;
   Program4.Spare3H3 := 0;
   Program4.Spare59 := 0;
   Program4.Spare60 := 0;
   Program4.Spare61 := 380;
   Program4.Spare62 := 2800;
   Program4.Spare63 := 0;
   Program4.Overlap3_4 := 100;
   Program4.Height4 := 100;
   Program4.Landmark4 := FALSE;
   Program4.Lifter4 := FALSE;
   Program4.SpareBit1H4 := FALSE;
   Program4.Airblower4 := TRUE;
   Program4.NextStep4 := TRUE;
   Program4.PressureP4 := TRUE;
   Program4.SpareByte2H4 := 16#00;
   Program4.Revolution4 := 3;
   Program4.RopeUnit4_1 := 16#02;
   Program4.RopeUnit4_2 := 16#02;
   Program4.FilmForce4 := 30;
   Program4.FilmPrestretch4 := 200;
   Program4.Spare3H4 := 0;
   Program4.Spare64 := 0;
   Program4.Spare65 := 0;
   Program4.Spare66 := 0;
   Program4.Spare67 := 0;
   Program4.Spare68 := 0;
   Program4.Overlap4_5 := 0;
   Program4.Height5 := 50;
   Program4.Landmark5 := FALSE;
   Program4.Lifter5 := FALSE;
   Program4.SpareBit1H5 := FALSE;
   Program4.Airblower5 := TRUE;
   Program4.NextStep5 := FALSE;
   Program4.PressureP5 := FALSE;
   Program4.SpareByte2H5 := 16#00;
   Program4.Revolution5 := 1;
   Program4.RopeUnit5_1 := 16#01;
   Program4.RopeUnit5_2 := 16#01;
   Program4.FilmForce5 := 30;
   Program4.FilmPrestretch5 := 200;
   Program4.Spare3H5 := 0;
   Program4.Spare69 := 0;
   Program4.Spare70 := 0;
   Program4.Spare71 := 0;
   Program4.Spare72 := 0;
   Program4.Spare73 := 0;
   Program4.Overlap5_6 := 100;
   Program4.Height6 := 50;
   Program4.Landmark6 := FALSE;
   Program4.Lifter6 := FALSE;
   Program4.SpareBit1H6 := FALSE;
   Program4.Airblower6 := TRUE;
   Program4.NextStep6 := FALSE;
   Program4.PressureP6 := FALSE;
   Program4.SpareByte2H6 := 16#00;
   Program4.Revolution6 := 2;
   Program4.RopeUnit6_1 := 16#02;
   Program4.RopeUnit6_2 := 16#01;
   Program4.FilmForce6 := 20;
   Program4.FilmPrestretch6 := 200;
   Program4.Spare3H6 := 0;
   Program4.Spare74 := 0;
   Program4.Spare75 := 0;
   Program4.Spare76 := 0;
   Program4.Spare77 := 0;
   Program4.Spare78 := 0;
   Program4.Overlap6_7 := 0;
   Program4.Height7 := 0;
   Program4.Landmark7 := FALSE;
   Program4.Lifter7 := FALSE;
   Program4.SpareBit1H7 := FALSE;
   Program4.Airblower7 := FALSE;
   Program4.NextStep7 := TRUE;
   Program4.PressureP7 := FALSE;
   Program4.SpareByte2H7 := 16#00;
   Program4.Revolution7 := 1;
   Program4.RopeUnit7_1 := 16#01;
   Program4.RopeUnit7_2 := 16#01;
   Program4.FilmForce7 := 0;
   Program4.FilmPrestretch7 := 100;
   Program4.Spare3H7 := 0;
   Program4.Spare79 := 0;
   Program4.Spare80 := 0;
   Program4.Spare81 := 0;
   Program4.Spare82 := 0;
   Program4.Spare83 := 0;
   Program4.Overlap7_8 := 0;
   Program4.Height8 := 0;
   Program4.Landmark8 := FALSE;
   Program4.Lifter8 := FALSE;
   Program4.SpareBit1H8 := FALSE;
   Program4.Airblower8 := FALSE;
   Program4.NextStep8 := TRUE;
   Program4.PressureP8 := FALSE;
   Program4.SpareByte2H8 := 16#00;
   Program4.Revolution8 := 1;
   Program4.RopeUnit8_1 := 16#01;
   Program4.RopeUnit8_2 := 16#01;
   Program4.FilmForce8 := 0;
   Program4.FilmPrestretch8 := 100;
   Program4.Spare3H8 := 0;
   Program4.Spare84 := 0;
   Program4.Spare85 := 0;
   Program4.Spare86 := 0;
   Program4.Spare87 := 0;
   Program4.Spare88 := 0;
   Program4.Overlap8_9 := 0;
   Program4.Height9 := 0;
   Program4.Landmark9 := FALSE;
   Program4.Lifter9 := FALSE;
   Program4.SpareBit1H9 := FALSE;
   Program4.Airblower9 := FALSE;
   Program4.NextStep9 := TRUE;
   Program4.PressureP9 := FALSE;
   Program4.SpareByte2H9 := 16#00;
   Program4.Revolution9 := 1;
   Program4.RopeUnit9_1 := 16#01;
   Program4.RopeUnit9_2 := 16#01;
   Program4.FilmForce9 := 0;
   Program4.FilmPrestretch9 := 100;
   Program4.Spare3H9 := 0;
   Program4.Spare89 := 0;
   Program4.Spare90 := 0;
   Program4.Spare91 := 0;
   Program4.Spare92 := 0;
   Program4.Spare93 := 0;
   Program4.Overlap9_10 := 0;
   Program4.Height10 := 0;
   Program4.Landmark10 := FALSE;
   Program4.Lifter10 := FALSE;
   Program4.SpareBit1H10 := FALSE;
   Program4.Airblower10 := FALSE;
   Program4.NextStep10 := FALSE;
   Program4.PressureP10 := FALSE;
   Program4.SpareByte2H10 := 16#00;
   Program4.Revolution10 := 1;
   Program4.RopeUnit10_1 := 16#01;
   Program4.RopeUnit10_2 := 16#01;
   Program4.FilmForce10 := 0;
   Program4.FilmPrestretch10 := 100;
   Program4.Spare3H10 := 0;
   Program4.Spare94 := 0;
   Program4.Spare95 := 0;
   Program4.Spare96 := 0;
   Program4.Spare97 := 0;
   Program4.Spare98 := 0;
   Program4.Overlap10_11 := 0;
   Program4.Height11 := 0;
   Program4.Landmark11 := FALSE;
   Program4.Lifter11 := FALSE;
   Program4.SpareBit1H11 := FALSE;
   Program4.Airblower11 := FALSE;
   Program4.NextStep11 := TRUE;
   Program4.PressureP11 := FALSE;
   Program4.SpareByte2H11 := 16#00;
   Program4.Revolution11 := 1;
   Program4.RopeUnit11_1 := 16#01;
   Program4.RopeUnit11_2 := 16#01;
   Program4.FilmForce11 := 0;
   Program4.FilmPrestretch11 := 100;
   Program4.Spare3H11 := 0;
   Program4.Spare99 := 0;
   Program4.Spare100 := 0;
   Program4.Spare101 := 0;
   Program4.Spare102 := 0;
   Program4.Spare103 := 0;
   Program4.Overlap11_12 := 0;
   Program4.Height12 := 0;
   Program4.Landmark12 := FALSE;
   Program4.Lifter12 := FALSE;
   Program4.SpareBit1H12 := FALSE;
   Program4.Airblower12 := FALSE;
   Program4.NextStep12 := FALSE;
   Program4.PressureP12 := FALSE;
   Program4.SpareByte2H12 := 16#00;
   Program4.Revolution12 := 1;
   Program4.RopeUnit12_1 := 16#01;
   Program4.RopeUnit12_2 := 16#01;
   Program4.FilmForce12 := 0;
   Program4.FilmPrestretch12 := 100;
   Program4.Spare3H12 := 0;
   Program4.Spare104 := 0;
   Program4.Spare105 := 0;
   Program4.Spare106 := 0;
   Program4.Spare107 := 0;
   Program4.Spare108 := 0;
END_DATA_BLOCK

DATA_BLOCK "DB247_Program3"   // DB247
{ S7_Optimized_Access := 'FALSE' }
AUTHOR : Robopac
VERSION : 0.0
// stored: AutoNumber false, IsOnlyStoredInLoadMemory false, IsWriteProtectedInAS false
   VAR RETAIN
      Program3 { S7_SetPoint := 'True'} : "DatiProgramma";
   END_VAR
BEGIN
   Program3.Wrapping := TRUE;
   Program3.TopLenght := 500;
   Program3.TopRelease := 0;
   Program3.TopDown := 0;
   Program3.Top := 4;
   Program3.PressurePTime := 0;
   Program3.LifterTime := 0;
   Program3.RevOverContrast := 1;
   Program3.RopeEndCycle := 16#01;
   Program3.Spare4 := 16#01;
   Program3.RopeTime := 1500;
   Program3.RevOverClamp := 1;
   Program3.FilmForceFinalRev := 20;
   Program3.FilmPrestretchFinalRev := 100;
   Program3.ArmSpeed := 90;
   Program3.CarriageDown4Top := 500;
   Program3.TopDownTime := 1500;
   Program3.LapsUnderTop := 0;
   Program3.Spare6 := 0;
   Program3.Spare7 := 0;
   Program3.Spare8 := 0;
   Program3.Spare9 := 0;
   Program3.Spare10 := 0;
   Program3.Spare11 := 0;
   Program3.Spare12 := 0;
   Program3.Overlap0_1 := 0;
   Program3.Height1 := 120;
   Program3.Landmark1 := FALSE;
   Program3.Lifter1 := FALSE;
   Program3.SpareBit1H1 := FALSE;
   Program3.Airblower1 := TRUE;
   Program3.NextStep1 := TRUE;
   Program3.PressureP1 := TRUE;
   Program3.SpareByte2H1 := 16#00;
   Program3.Revolution1 := 1;
   Program3.RopeUnit1_1 := 16#01;
   Program3.RopeUnit1_2 := 16#01;
   Program3.FilmForce1 := 5;
   Program3.FilmPrestretch1 := 200;
   Program3.Spare3H1 := 0;
   Program3.Spare49 := 0;
   Program3.Spare50 := 0;
   Program3.Spare51 := 0;
   Program3.Spare52 := 0;
   Program3.Spare53 := 0;
   Program3.Overlap1_2 := 0;
   Program3.Height2 := 60;
   Program3.Landmark2 := FALSE;
   Program3.Lifter2 := FALSE;
   Program3.SpareBit1H2 := FALSE;
   Program3.Airblower2 := TRUE;
   Program3.NextStep2 := TRUE;
   Program3.PressureP2 := TRUE;
   Program3.SpareByte2H2 := 16#00;
   Program3.Revolution2 := 3;
   Program3.RopeUnit2_1 := 16#01;
   Program3.RopeUnit2_2 := 16#01;
   Program3.FilmForce2 := 10;
   Program3.FilmPrestretch2 := 200;
   Program3.Spare3H2 := 0;
   Program3.Spare54 := 0;
   Program3.Spare55 := 0;
   Program3.Spare56 := 0;
   Program3.Spare57 := 0;
   Program3.Spare58 := 0;
   Program3.Overlap2_3 := 100;
   Program3.Height3 := 120;
   Program3.Landmark3 := FALSE;
   Program3.Lifter3 := FALSE;
   Program3.SpareBit1H3 := FALSE;
   Program3.Airblower3 := TRUE;
   Program3.NextStep3 := TRUE;
   Program3.PressureP3 := TRUE;
   Program3.SpareByte2H3 := 16#00;
   Program3.Revolution3 := 2;
   Program3.RopeUnit3_1 := 16#01;
   Program3.RopeUnit3_2 := 16#01;
   Program3.FilmForce3 := 5;
   Program3.FilmPrestretch3 := 200;
   Program3.Spare3H3 := 0;
   Program3.Spare59 := 0;
   Program3.Spare60 := 0;
   Program3.Spare61 := 380;
   Program3.Spare62 := 2800;
   Program3.Spare63 := 0;
   Program3.Overlap3_4 := 200;
   Program3.Height4 := 120;
   Program3.Landmark4 := FALSE;
   Program3.Lifter4 := FALSE;
   Program3.SpareBit1H4 := FALSE;
   Program3.Airblower4 := TRUE;
   Program3.NextStep4 := TRUE;
   Program3.PressureP4 := TRUE;
   Program3.SpareByte2H4 := 16#00;
   Program3.Revolution4 := 1;
   Program3.RopeUnit4_1 := 16#01;
   Program3.RopeUnit4_2 := 16#01;
   Program3.FilmForce4 := 20;
   Program3.FilmPrestretch4 := 200;
   Program3.Spare3H4 := 0;
   Program3.Spare64 := 0;
   Program3.Spare65 := 0;
   Program3.Spare66 := 0;
   Program3.Spare67 := 0;
   Program3.Spare68 := 0;
   Program3.Overlap4_5 := 200;
   Program3.Height5 := -150;
   Program3.Landmark5 := TRUE;
   Program3.Lifter5 := FALSE;
   Program3.SpareBit1H5 := FALSE;
   Program3.Airblower5 := FALSE;
   Program3.NextStep5 := TRUE;
   Program3.PressureP5 := FALSE;
   Program3.SpareByte2H5 := 16#00;
   Program3.Revolution5 := 1;
   Program3.RopeUnit5_1 := 16#01;
   Program3.RopeUnit5_2 := 16#01;
   Program3.FilmForce5 := 20;
   Program3.FilmPrestretch5 := 200;
   Program3.Spare3H5 := 0;
   Program3.Spare69 := 0;
   Program3.Spare70 := 0;
   Program3.Spare71 := 0;
   Program3.Spare72 := 0;
   Program3.Spare73 := 0;
   Program3.Overlap5_6 := 100;
   Program3.Height6 := 0;
   Program3.Landmark6 := FALSE;
   Program3.Lifter6 := FALSE;
   Program3.SpareBit1H6 := FALSE;
   Program3.Airblower6 := FALSE;
   Program3.NextStep6 := FALSE;
   Program3.PressureP6 := FALSE;
   Program3.SpareByte2H6 := 16#00;
   Program3.Revolution6 := 1;
   Program3.RopeUnit6_1 := 16#01;
   Program3.RopeUnit6_2 := 16#01;
   Program3.FilmForce6 := 30;
   Program3.FilmPrestretch6 := 200;
   Program3.Spare3H6 := 0;
   Program3.Spare74 := 0;
   Program3.Spare75 := 0;
   Program3.Spare76 := 0;
   Program3.Spare77 := 0;
   Program3.Spare78 := 0;
   Program3.Overlap6_7 := 0;
   Program3.Height7 := 0;
   Program3.Landmark7 := FALSE;
   Program3.Lifter7 := FALSE;
   Program3.SpareBit1H7 := FALSE;
   Program3.Airblower7 := FALSE;
   Program3.NextStep7 := TRUE;
   Program3.PressureP7 := FALSE;
   Program3.SpareByte2H7 := 16#00;
   Program3.Revolution7 := 1;
   Program3.RopeUnit7_1 := 16#01;
   Program3.RopeUnit7_2 := 16#01;
   Program3.FilmForce7 := 0;
   Program3.FilmPrestretch7 := 100;
   Program3.Spare3H7 := 0;
   Program3.Spare79 := 0;
   Program3.Spare80 := 0;
   Program3.Spare81 := 0;
   Program3.Spare82 := 0;
   Program3.Spare83 := 0;
   Program3.Overlap7_8 := 0;
   Program3.Height8 := 0;
   Program3.Landmark8 := FALSE;
   Program3.Lifter8 := FALSE;
   Program3.SpareBit1H8 := FALSE;
   Program3.Airblower8 := FALSE;
   Program3.NextStep8 := TRUE;
   Program3.PressureP8 := FALSE;
   Program3.SpareByte2H8 := 16#00;
   Program3.Revolution8 := 1;
   Program3.RopeUnit8_1 := 16#01;
   Program3.RopeUnit8_2 := 16#01;
   Program3.FilmForce8 := 0;
   Program3.FilmPrestretch8 := 100;
   Program3.Spare3H8 := 0;
   Program3.Spare84 := 0;
   Program3.Spare85 := 0;
   Program3.Spare86 := 0;
   Program3.Spare87 := 0;
   Program3.Spare88 := 0;
   Program3.Overlap8_9 := 0;
   Program3.Height9 := 0;
   Program3.Landmark9 := FALSE;
   Program3.Lifter9 := FALSE;
   Program3.SpareBit1H9 := FALSE;
   Program3.Airblower9 := FALSE;
   Program3.NextStep9 := TRUE;
   Program3.PressureP9 := FALSE;
   Program3.SpareByte2H9 := 16#00;
   Program3.Revolution9 := 1;
   Program3.RopeUnit9_1 := 16#01;
   Program3.RopeUnit9_2 := 16#01;
   Program3.FilmForce9 := 0;
   Program3.FilmPrestretch9 := 100;
   Program3.Spare3H9 := 0;
   Program3.Spare89 := 0;
   Program3.Spare90 := 0;
   Program3.Spare91 := 0;
   Program3.Spare92 := 0;
   Program3.Spare93 := 0;
   Program3.Overlap9_10 := 0;
   Program3.Height10 := 0;
   Program3.Landmark10 := FALSE;
   Program3.Lifter10 := FALSE;
   Program3.SpareBit1H10 := FALSE;
   Program3.Airblower10 := FALSE;
   Program3.NextStep10 := FALSE;
   Program3.PressureP10 := FALSE;
   Program3.SpareByte2H10 := 16#00;
   Program3.Revolution10 := 1;
   Program3.RopeUnit10_1 := 16#01;
   Program3.RopeUnit10_2 := 16#01;
   Program3.FilmForce10 := 0;
   Program3.FilmPrestretch10 := 100;
   Program3.Spare3H10 := 0;
   Program3.Spare94 := 0;
   Program3.Spare95 := 0;
   Program3.Spare96 := 0;
   Program3.Spare97 := 0;
   Program3.Spare98 := 0;
   Program3.Overlap10_11 := 0;
   Program3.Height11 := 0;
   Program3.Landmark11 := FALSE;
   Program3.Lifter11 := FALSE;
   Program3.SpareBit1H11 := FALSE;
   Program3.Airblower11 := FALSE;
   Program3.NextStep11 := TRUE;
   Program3.PressureP11 := FALSE;
   Program3.SpareByte2H11 := 16#00;
   Program3.Revolution11 := 1;
   Program3.RopeUnit11_1 := 16#01;
   Program3.RopeUnit11_2 := 16#01;
   Program3.FilmForce11 := 0;
   Program3.FilmPrestretch11 := 100;
   Program3.Spare3H11 := 0;
   Program3.Spare99 := 0;
   Program3.Spare100 := 0;
   Program3.Spare101 := 0;
   Program3.Spare102 := 0;
   Program3.Spare103 := 0;
   Program3.Overlap11_12 := 0;
   Program3.Height12 := 0;
   Program3.Landmark12 := FALSE;
   Program3.Lifter12 := FALSE;
   Program3.SpareBit1H12 := FALSE;
   Program3.Airblower12 := FALSE;
   Program3.NextStep12 := FALSE;
   Program3.PressureP12 := FALSE;
   Program3.SpareByte2H12 := 16#00;
   Program3.Revolution12 := 1;
   Program3.RopeUnit12_1 := 16#01;
   Program3.RopeUnit12_2 := 16#01;
   Program3.FilmForce12 := 0;
   Program3.FilmPrestretch12 := 100;
   Program3.Spare3H12 := 0;
   Program3.Spare104 := 0;
   Program3.Spare105 := 0;
   Program3.Spare106 := 0;
   Program3.Spare107 := 0;
   Program3.Spare108 := 0;
END_DATA_BLOCK

DATA_BLOCK "DB248_Program2"   // DB248
{ S7_Optimized_Access := 'FALSE' }
AUTHOR : Robopac
VERSION : 0.0
// stored: AutoNumber false, IsOnlyStoredInLoadMemory false, IsWriteProtectedInAS false
   VAR RETAIN
      Program2 { S7_SetPoint := 'True'} : "DatiProgramma";
   END_VAR
BEGIN
   Program2.Wrapping := TRUE;
   Program2.TopLenght := 500;
   Program2.TopRelease := 0;
   Program2.TopDown := 0;
   Program2.Top := 4;
   Program2.PressurePTime := 0;
   Program2.LifterTime := 0;
   Program2.RevOverContrast := 1;
   Program2.RopeEndCycle := 16#01;
   Program2.Spare4 := 16#01;
   Program2.RopeTime := 1500;
   Program2.RevOverClamp := 1;
   Program2.FilmForceFinalRev := 35;
   Program2.FilmPrestretchFinalRev := 100;
   Program2.ArmSpeed := 85;
   Program2.CarriageDown4Top := 500;
   Program2.TopDownTime := 1500;
   Program2.LapsUnderTop := 0;
   Program2.Spare6 := 0;
   Program2.Spare7 := 0;
   Program2.Spare8 := 0;
   Program2.Spare9 := 0;
   Program2.Spare10 := 0;
   Program2.Spare11 := 0;
   Program2.Spare12 := 0;
   Program2.Overlap0_1 := 0;
   Program2.Height1 := 180;
   Program2.Landmark1 := FALSE;
   Program2.Lifter1 := FALSE;
   Program2.SpareBit1H1 := FALSE;
   Program2.Airblower1 := TRUE;
   Program2.NextStep1 := TRUE;
   Program2.PressureP1 := TRUE;
   Program2.SpareByte2H1 := 16#00;
   Program2.Revolution1 := 1;
   Program2.RopeUnit1_1 := 16#01;
   Program2.RopeUnit1_2 := 16#01;
   Program2.FilmForce1 := 5;
   Program2.FilmPrestretch1 := 200;
   Program2.Spare3H1 := 0;
   Program2.Spare49 := 0;
   Program2.Spare50 := 0;
   Program2.Spare51 := 0;
   Program2.Spare52 := 0;
   Program2.Spare53 := 0;
   Program2.Overlap1_2 := 200;
   Program2.Height2 := -100;
   Program2.Landmark2 := TRUE;
   Program2.Lifter2 := FALSE;
   Program2.SpareBit1H2 := FALSE;
   Program2.Airblower2 := TRUE;
   Program2.NextStep2 := TRUE;
   Program2.PressureP2 := TRUE;
   Program2.SpareByte2H2 := 16#00;
   Program2.Revolution2 := 2;
   Program2.RopeUnit2_1 := 16#01;
   Program2.RopeUnit2_2 := 16#01;
   Program2.FilmForce2 := 20;
   Program2.FilmPrestretch2 := 200;
   Program2.Spare3H2 := 0;
   Program2.Spare54 := 0;
   Program2.Spare55 := 0;
   Program2.Spare56 := 0;
   Program2.Spare57 := 0;
   Program2.Spare58 := 0;
   Program2.Overlap2_3 := 200;
   Program2.Height3 := 80;
   Program2.Landmark3 := FALSE;
   Program2.Lifter3 := FALSE;
   Program2.SpareBit1H3 := FALSE;
   Program2.Airblower3 := TRUE;
   Program2.NextStep3 := TRUE;
   Program2.PressureP3 := TRUE;
   Program2.SpareByte2H3 := 16#00;
   Program2.Revolution3 := 2;
   Program2.RopeUnit3_1 := 16#01;
   Program2.RopeUnit3_2 := 16#01;
   Program2.FilmForce3 := 10;
   Program2.FilmPrestretch3 := 200;
   Program2.Spare3H3 := 0;
   Program2.Spare59 := 0;
   Program2.Spare60 := 0;
   Program2.Spare61 := 380;
   Program2.Spare62 := 2800;
   Program2.Spare63 := 0;
   Program2.Overlap3_4 := 200;
   Program2.Height4 := 120;
   Program2.Landmark4 := FALSE;
   Program2.Lifter4 := FALSE;
   Program2.SpareBit1H4 := FALSE;
   Program2.Airblower4 := TRUE;
   Program2.NextStep4 := TRUE;
   Program2.PressureP4 := TRUE;
   Program2.SpareByte2H4 := 16#00;
   Program2.Revolution4 := 2;
   Program2.RopeUnit4_1 := 16#02;
   Program2.RopeUnit4_2 := 16#02;
   Program2.FilmForce4 := 20;
   Program2.FilmPrestretch4 := 200;
   Program2.Spare3H4 := 0;
   Program2.Spare64 := 0;
   Program2.Spare65 := 0;
   Program2.Spare66 := 0;
   Program2.Spare67 := 0;
   Program2.Spare68 := 0;
   Program2.Overlap4_5 := 200;
   Program2.Height5 := 90;
   Program2.Landmark5 := FALSE;
   Program2.Lifter5 := FALSE;
   Program2.SpareBit1H5 := FALSE;
   Program2.Airblower5 := TRUE;
   Program2.NextStep5 := FALSE;
   Program2.PressureP5 := FALSE;
   Program2.SpareByte2H5 := 16#00;
   Program2.Revolution5 := 1;
   Program2.RopeUnit5_1 := 16#01;
   Program2.RopeUnit5_2 := 16#01;
   Program2.FilmForce5 := 20;
   Program2.FilmPrestretch5 := 200;
   Program2.Spare3H5 := 0;
   Program2.Spare69 := 0;
   Program2.Spare70 := 0;
   Program2.Spare71 := 0;
   Program2.Spare72 := 0;
   Program2.Spare73 := 0;
   Program2.Overlap5_6 := 300;
   Program2.Height6 := 120;
   Program2.Landmark6 := FALSE;
   Program2.Lifter6 := FALSE;
   Program2.SpareBit1H6 := FALSE;
   Program2.Airblower6 := TRUE;
   Program2.NextStep6 := FALSE;
   Program2.PressureP6 := FALSE;
   Program2.SpareByte2H6 := 16#00;
   Program2.Revolution6 := 1;
   Program2.RopeUnit6_1 := 16#01;
   Program2.RopeUnit6_2 := 16#01;
   Program2.FilmForce6 := 20;
   Program2.FilmPrestretch6 := 200;
   Program2.Spare3H6 := 0;
   Program2.Spare74 := 0;
   Program2.Spare75 := 0;
   Program2.Spare76 := 0;
   Program2.Spare77 := 0;
   Program2.Spare78 := 0;
   Program2.Overlap6_7 := 0;
   Program2.Height7 := 0;
   Program2.Landmark7 := FALSE;
   Program2.Lifter7 := FALSE;
   Program2.SpareBit1H7 := FALSE;
   Program2.Airblower7 := FALSE;
   Program2.NextStep7 := TRUE;
   Program2.PressureP7 := FALSE;
   Program2.SpareByte2H7 := 16#00;
   Program2.Revolution7 := 1;
   Program2.RopeUnit7_1 := 16#01;
   Program2.RopeUnit7_2 := 16#01;
   Program2.FilmForce7 := 0;
   Program2.FilmPrestretch7 := 100;
   Program2.Spare3H7 := 0;
   Program2.Spare79 := 0;
   Program2.Spare80 := 0;
   Program2.Spare81 := 0;
   Program2.Spare82 := 0;
   Program2.Spare83 := 0;
   Program2.Overlap7_8 := 0;
   Program2.Height8 := 0;
   Program2.Landmark8 := FALSE;
   Program2.Lifter8 := FALSE;
   Program2.SpareBit1H8 := FALSE;
   Program2.Airblower8 := FALSE;
   Program2.NextStep8 := TRUE;
   Program2.PressureP8 := FALSE;
   Program2.SpareByte2H8 := 16#00;
   Program2.Revolution8 := 1;
   Program2.RopeUnit8_1 := 16#01;
   Program2.RopeUnit8_2 := 16#01;
   Program2.FilmForce8 := 0;
   Program2.FilmPrestretch8 := 100;
   Program2.Spare3H8 := 0;
   Program2.Spare84 := 0;
   Program2.Spare85 := 0;
   Program2.Spare86 := 0;
   Program2.Spare87 := 0;
   Program2.Spare88 := 0;
   Program2.Overlap8_9 := 0;
   Program2.Height9 := 0;
   Program2.Landmark9 := FALSE;
   Program2.Lifter9 := FALSE;
   Program2.SpareBit1H9 := FALSE;
   Program2.Airblower9 := FALSE;
   Program2.NextStep9 := TRUE;
   Program2.PressureP9 := FALSE;
   Program2.SpareByte2H9 := 16#00;
   Program2.Revolution9 := 1;
   Program2.RopeUnit9_1 := 16#01;
   Program2.RopeUnit9_2 := 16#01;
   Program2.FilmForce9 := 0;
   Program2.FilmPrestretch9 := 100;
   Program2.Spare3H9 := 0;
   Program2.Spare89 := 0;
   Program2.Spare90 := 0;
   Program2.Spare91 := 0;
   Program2.Spare92 := 0;
   Program2.Spare93 := 0;
   Program2.Overlap9_10 := 0;
   Program2.Height10 := 0;
   Program2.Landmark10 := FALSE;
   Program2.Lifter10 := FALSE;
   Program2.SpareBit1H10 := FALSE;
   Program2.Airblower10 := FALSE;
   Program2.NextStep10 := FALSE;
   Program2.PressureP10 := FALSE;
   Program2.SpareByte2H10 := 16#00;
   Program2.Revolution10 := 1;
   Program2.RopeUnit10_1 := 16#01;
   Program2.RopeUnit10_2 := 16#01;
   Program2.FilmForce10 := 0;
   Program2.FilmPrestretch10 := 100;
   Program2.Spare3H10 := 0;
   Program2.Spare94 := 0;
   Program2.Spare95 := 0;
   Program2.Spare96 := 0;
   Program2.Spare97 := 0;
   Program2.Spare98 := 0;
   Program2.Overlap10_11 := 0;
   Program2.Height11 := 0;
   Program2.Landmark11 := FALSE;
   Program2.Lifter11 := FALSE;
   Program2.SpareBit1H11 := FALSE;
   Program2.Airblower11 := FALSE;
   Program2.NextStep11 := TRUE;
   Program2.PressureP11 := FALSE;
   Program2.SpareByte2H11 := 16#00;
   Program2.Revolution11 := 1;
   Program2.RopeUnit11_1 := 16#01;
   Program2.RopeUnit11_2 := 16#01;
   Program2.FilmForce11 := 0;
   Program2.FilmPrestretch11 := 100;
   Program2.Spare3H11 := 0;
   Program2.Spare99 := 0;
   Program2.Spare100 := 0;
   Program2.Spare101 := 0;
   Program2.Spare102 := 0;
   Program2.Spare103 := 0;
   Program2.Overlap11_12 := 0;
   Program2.Height12 := 0;
   Program2.Landmark12 := FALSE;
   Program2.Lifter12 := FALSE;
   Program2.SpareBit1H12 := FALSE;
   Program2.Airblower12 := FALSE;
   Program2.NextStep12 := FALSE;
   Program2.PressureP12 := FALSE;
   Program2.SpareByte2H12 := 16#00;
   Program2.Revolution12 := 1;
   Program2.RopeUnit12_1 := 16#01;
   Program2.RopeUnit12_2 := 16#01;
   Program2.FilmForce12 := 0;
   Program2.FilmPrestretch12 := 100;
   Program2.Spare3H12 := 0;
   Program2.Spare104 := 0;
   Program2.Spare105 := 0;
   Program2.Spare106 := 0;
   Program2.Spare107 := 0;
   Program2.Spare108 := 0;
END_DATA_BLOCK

DATA_BLOCK "DB249_Program1"   // DB249
{ S7_Optimized_Access := 'FALSE' }
AUTHOR : Robopac
VERSION : 0.0
// stored: AutoNumber false, IsOnlyStoredInLoadMemory false, IsWriteProtectedInAS false
   VAR RETAIN
      Program1 { S7_SetPoint := 'True'} : "DatiProgramma";
   END_VAR
BEGIN
   Program1.Wrapping := TRUE;
   Program1.TopLenght := 500;
   Program1.TopRelease := 0;
   Program1.TopDown := 0;
   Program1.Top := 4;
   Program1.PressurePTime := 0;
   Program1.LifterTime := 0;
   Program1.RevOverContrast := 1;
   Program1.RopeEndCycle := 16#02;
   Program1.Spare4 := 16#01;
   Program1.RopeTime := 1500;
   Program1.RevOverClamp := 1;
   Program1.FilmForceFinalRev := 25;
   Program1.FilmPrestretchFinalRev := 100;
   Program1.ArmSpeed := 87;
   Program1.CarriageDown4Top := 500;
   Program1.TopDownTime := 1500;
   Program1.LapsUnderTop := 0;
   Program1.Spare6 := 0;
   Program1.Spare7 := 0;
   Program1.Spare8 := 0;
   Program1.Spare9 := 0;
   Program1.Spare10 := 0;
   Program1.Spare11 := 0;
   Program1.Spare12 := 0;
   Program1.Overlap0_1 := 0;
   Program1.Height1 := 120;
   Program1.Landmark1 := FALSE;
   Program1.Lifter1 := FALSE;
   Program1.SpareBit1H1 := FALSE;
   Program1.Airblower1 := TRUE;
   Program1.NextStep1 := TRUE;
   Program1.PressureP1 := TRUE;
   Program1.SpareByte2H1 := 16#00;
   Program1.Revolution1 := 1;
   Program1.RopeUnit1_1 := 16#03;
   Program1.RopeUnit1_2 := 16#01;
   Program1.FilmForce1 := 5;
   Program1.FilmPrestretch1 := 200;
   Program1.Spare3H1 := 0;
   Program1.Spare49 := 0;
   Program1.Spare50 := 0;
   Program1.Spare51 := 0;
   Program1.Spare52 := 0;
   Program1.Spare53 := 0;
   Program1.Overlap1_2 := 0;
   Program1.Height2 := 85;
   Program1.Landmark2 := FALSE;
   Program1.Lifter2 := FALSE;
   Program1.SpareBit1H2 := FALSE;
   Program1.Airblower2 := TRUE;
   Program1.NextStep2 := TRUE;
   Program1.PressureP2 := TRUE;
   Program1.SpareByte2H2 := 16#00;
   Program1.Revolution2 := 3;
   Program1.RopeUnit2_1 := 16#01;
   Program1.RopeUnit2_2 := 16#01;
   Program1.FilmForce2 := 15;
   Program1.FilmPrestretch2 := 200;
   Program1.Spare3H2 := 0;
   Program1.Spare54 := 0;
   Program1.Spare55 := 0;
   Program1.Spare56 := 0;
   Program1.Spare57 := 0;
   Program1.Spare58 := 0;
   Program1.Overlap2_3 := 300;
   Program1.Height3 := 110;
   Program1.Landmark3 := FALSE;
   Program1.Lifter3 := FALSE;
   Program1.SpareBit1H3 := FALSE;
   Program1.Airblower3 := TRUE;
   Program1.NextStep3 := TRUE;
   Program1.PressureP3 := TRUE;
   Program1.SpareByte2H3 := 16#00;
   Program1.Revolution3 := 2;
   Program1.RopeUnit3_1 := 16#03;
   Program1.RopeUnit3_2 := 16#03;
   Program1.FilmForce3 := 20;
   Program1.FilmPrestretch3 := 200;
   Program1.Spare3H3 := 0;
   Program1.Spare59 := 0;
   Program1.Spare60 := 0;
   Program1.Spare61 := 380;
   Program1.Spare62 := 2800;
   Program1.Spare63 := 0;
   Program1.Overlap3_4 := 100;
   Program1.Height4 := -100;
   Program1.Landmark4 := TRUE;
   Program1.Lifter4 := FALSE;
   Program1.SpareBit1H4 := FALSE;
   Program1.Airblower4 := FALSE;
   Program1.NextStep4 := TRUE;
   Program1.PressureP4 := TRUE;
   Program1.SpareByte2H4 := 16#00;
   Program1.Revolution4 := 1;
   Program1.RopeUnit4_1 := 16#01;
   Program1.RopeUnit4_2 := 16#01;
   Program1.FilmForce4 := 18;
   Program1.FilmPrestretch4 := 200;
   Program1.Spare3H4 := 0;
   Program1.Spare64 := 0;
   Program1.Spare65 := 0;
   Program1.Spare66 := 0;
   Program1.Spare67 := 0;
   Program1.Spare68 := 0;
   Program1.Overlap4_5 := 100;
   Program1.Height5 := 60;
   Program1.Landmark5 := FALSE;
   Program1.Lifter5 := FALSE;
   Program1.SpareBit1H5 := FALSE;
   Program1.Airblower5 := TRUE;
   Program1.NextStep5 := TRUE;
   Program1.PressureP5 := FALSE;
   Program1.SpareByte2H5 := 16#00;
   Program1.Revolution5 := 1;
   Program1.RopeUnit5_1 := 16#01;
   Program1.RopeUnit5_2 := 16#01;
   Program1.FilmForce5 := 25;
   Program1.FilmPrestretch5 := 200;
   Program1.Spare3H5 := 0;
   Program1.Spare69 := 0;
   Program1.Spare70 := 0;
   Program1.Spare71 := 0;
   Program1.Spare72 := 0;
   Program1.Spare73 := 0;
   Program1.Overlap5_6 := 100;
   Program1.Height6 := 40;
   Program1.Landmark6 := FALSE;
   Program1.Lifter6 := FALSE;
   Program1.SpareBit1H6 := FALSE;
   Program1.Airblower6 := TRUE;
   Program1.NextStep6 := FALSE;
   Program1.PressureP6 := FALSE;
   Program1.SpareByte2H6 := 16#00;
   Program1.Revolution6 := 1;
   Program1.RopeUnit6_1 := 16#01;
   Program1.RopeUnit6_2 := 16#01;
   Program1.FilmForce6 := 15;
   Program1.FilmPrestretch6 := 200;
   Program1.Spare3H6 := 0;
   Program1.Spare74 := 0;
   Program1.Spare75 := 0;
   Program1.Spare76 := 0;
   Program1.Spare77 := 0;
   Program1.Spare78 := 0;
   Program1.Overlap6_7 := 0;
   Program1.Height7 := 0;
   Program1.Landmark7 := FALSE;
   Program1.Lifter7 := FALSE;
   Program1.SpareBit1H7 := FALSE;
   Program1.Airblower7 := FALSE;
   Program1.NextStep7 := TRUE;
   Program1.PressureP7 := FALSE;
   Program1.SpareByte2H7 := 16#00;
   Program1.Revolution7 := 1;
   Program1.RopeUnit7_1 := 16#01;
   Program1.RopeUnit7_2 := 16#01;
   Program1.FilmForce7 := 0;
   Program1.FilmPrestretch7 := 100;
   Program1.Spare3H7 := 0;
   Program1.Spare79 := 0;
   Program1.Spare80 := 0;
   Program1.Spare81 := 0;
   Program1.Spare82 := 0;
   Program1.Spare83 := 0;
   Program1.Overlap7_8 := 0;
   Program1.Height8 := 0;
   Program1.Landmark8 := FALSE;
   Program1.Lifter8 := FALSE;
   Program1.SpareBit1H8 := FALSE;
   Program1.Airblower8 := FALSE;
   Program1.NextStep8 := TRUE;
   Program1.PressureP8 := FALSE;
   Program1.SpareByte2H8 := 16#00;
   Program1.Revolution8 := 1;
   Program1.RopeUnit8_1 := 16#01;
   Program1.RopeUnit8_2 := 16#01;
   Program1.FilmForce8 := 0;
   Program1.FilmPrestretch8 := 100;
   Program1.Spare3H8 := 0;
   Program1.Spare84 := 0;
   Program1.Spare85 := 0;
   Program1.Spare86 := 0;
   Program1.Spare87 := 0;
   Program1.Spare88 := 0;
   Program1.Overlap8_9 := 0;
   Program1.Height9 := 0;
   Program1.Landmark9 := FALSE;
   Program1.Lifter9 := FALSE;
   Program1.SpareBit1H9 := FALSE;
   Program1.Airblower9 := FALSE;
   Program1.NextStep9 := TRUE;
   Program1.PressureP9 := FALSE;
   Program1.SpareByte2H9 := 16#00;
   Program1.Revolution9 := 1;
   Program1.RopeUnit9_1 := 16#01;
   Program1.RopeUnit9_2 := 16#01;
   Program1.FilmForce9 := 0;
   Program1.FilmPrestretch9 := 100;
   Program1.Spare3H9 := 0;
   Program1.Spare89 := 0;
   Program1.Spare90 := 0;
   Program1.Spare91 := 0;
   Program1.Spare92 := 0;
   Program1.Spare93 := 0;
   Program1.Overlap9_10 := 0;
   Program1.Height10 := 0;
   Program1.Landmark10 := FALSE;
   Program1.Lifter10 := FALSE;
   Program1.SpareBit1H10 := FALSE;
   Program1.Airblower10 := FALSE;
   Program1.NextStep10 := FALSE;
   Program1.PressureP10 := FALSE;
   Program1.SpareByte2H10 := 16#00;
   Program1.Revolution10 := 1;
   Program1.RopeUnit10_1 := 16#01;
   Program1.RopeUnit10_2 := 16#01;
   Program1.FilmForce10 := 0;
   Program1.FilmPrestretch10 := 100;
   Program1.Spare3H10 := 0;
   Program1.Spare94 := 0;
   Program1.Spare95 := 0;
   Program1.Spare96 := 0;
   Program1.Spare97 := 0;
   Program1.Spare98 := 0;
   Program1.Overlap10_11 := 0;
   Program1.Height11 := 0;
   Program1.Landmark11 := FALSE;
   Program1.Lifter11 := FALSE;
   Program1.SpareBit1H11 := FALSE;
   Program1.Airblower11 := FALSE;
   Program1.NextStep11 := TRUE;
   Program1.PressureP11 := FALSE;
   Program1.SpareByte2H11 := 16#00;
   Program1.Revolution11 := 1;
   Program1.RopeUnit11_1 := 16#01;
   Program1.RopeUnit11_2 := 16#01;
   Program1.FilmForce11 := 0;
   Program1.FilmPrestretch11 := 100;
   Program1.Spare3H11 := 0;
   Program1.Spare99 := 0;
   Program1.Spare100 := 0;
   Program1.Spare101 := 0;
   Program1.Spare102 := 0;
   Program1.Spare103 := 0;
   Program1.Overlap11_12 := 0;
   Program1.Height12 := 0;
   Program1.Landmark12 := FALSE;
   Program1.Lifter12 := FALSE;
   Program1.SpareBit1H12 := FALSE;
   Program1.Airblower12 := FALSE;
   Program1.NextStep12 := FALSE;
   Program1.PressureP12 := FALSE;
   Program1.SpareByte2H12 := 16#00;
   Program1.Revolution12 := 1;
   Program1.RopeUnit12_1 := 16#01;
   Program1.RopeUnit12_2 := 16#01;
   Program1.FilmForce12 := 0;
   Program1.FilmPrestretch12 := 100;
   Program1.Spare3H12 := 0;
   Program1.Spare104 := 0;
   Program1.Spare105 := 0;
   Program1.Spare106 := 0;
   Program1.Spare107 := 0;
   Program1.Spare108 := 0;
END_DATA_BLOCK

